LIN {X 0,Y 361.924,Z 605.401,A -85,B 0,C 180,E1 -12943.066,E2 -12943.066} C_VEL
LIN {X 0,Y 361.991,Z 605.395,A -85,B 0,C 180,E1 -12946.528,E2 -12946.528} C_VEL
LIN {X 0,Y 362.028,Z 605.391,A -85,B 0,C 180,E1 -12949.938,E2 -12949.938} C_VEL
LIN {X 0,Y 362.143,Z 605.376,A -85,B 0,C 180,E1 -12952.193,E2 -12952.193} C_VEL
LIN {X 0,Y 362.116,Z 605.378,A -85,B 0,C 180,E1 -12954.432,E2 -12954.432} C_VEL
LIN {X 0,Y 362.281,Z 605.357,A -85,B 0,C 180,E1 -12957.777,E2 -12957.777} C_VEL
LIN {X 0,Y 362.421,Z 605.339,A -85,B 0,C 180,E1 -12960.001,E2 -12960.001} C_VEL
LIN {X 0,Y 362.275,Z 605.357,A -85,B 0,C 180,E1 -12962.224,E2 -12962.224} C_VEL
LIN {X 0,Y 362.169,Z 605.369,A -85,B 0,C 180,E1 -12966.687,E2 -12966.687} C_VEL
LIN {X 0,Y 362.068,Z 605.384,A -85,B 0,C 180,E1 -12968.934,E2 -12968.934} C_VEL
LIN {X 0,Y 361.959,Z 605.395,A -85,B 0,C 180,E1 -12972.333,E2 -12972.333} C_VEL
LIN {X 0,Y 361.955,Z 605.398,A -85,B 0,C 180,E1 -12974.621,E2 -12974.621} C_VEL
LIN {X 0,Y 361.949,Z 605.397,A -85,B 0,C 180,E1 -12978.1,E2 -12978.1} C_VEL
LIN {X 0,Y 361.885,Z 605.403,A -85,B 0,C 180,E1 -12981.654,E2 -12981.654} C_VEL
LIN {X 0,Y 361.922,Z 605.398,A -85,B 0,C 180,E1 -12985.291,E2 -12985.291} C_VEL
LIN {X 0,Y 361.917,Z 605.399,A -85,B 0,C 180,E1 -12987.779,E2 -12987.779} C_VEL
LIN {X 0,Y 361.855,Z 605.403,A -85,B 0,C 180,E1 -12991.628,E2 -12991.628} C_VEL
LIN {X 0,Y 361.87,Z 605.404,A -85,B 0,C 180,E1 -12995.346,E2 -12995.346} C_VEL
LIN {X 0,Y 361.87,Z 605.406,A -85,B 0,C 180,E1 -12999.028,E2 -12999.028} C_VEL
LIN {X 0,Y 361.854,Z 605.41,A -85,B 0,C 180,E1 -13002.437,E2 -13002.437} C_VEL
LIN {X 0,Y 361.855,Z 605.41,A -85,B 0,C 180,E1 -13005.941,E2 -13005.941} C_VEL
LIN {X 0,Y 361.872,Z 605.412,A -85,B 0,C 180,E1 -13009.239,E2 -13009.239} C_VEL
LIN {X 0,Y 361.869,Z 605.41,A -85,B 0,C 180,E1 -13012.983,E2 -13012.983} C_VEL
LIN {X 0,Y 361.859,Z 605.415,A -85,B 0,C 180,E1 -13016.632,E2 -13016.632} C_VEL
LIN {X 0,Y 361.9,Z 605.535,A -85,B 0,C 180,E1 -13018.173,E2 -13018.173} C_VEL
LIN {X 0,Y 364.745,Z 617.624,A -85,B 0,C 180,E1 -13021.504,E2 -13021.504} C_VEL
LIN {X 0,Y 366.436,Z 626.629,A -85,B 0,C 180,E1 -13023.825,E2 -13023.825} C_VEL
LIN {X 0,Y 366.356,Z 630.226,A -85,B 0,C 180,E1 -13024.675,E2 -13024.675} C_VEL
LIN {X 0,Y 365,Z 642.315,A -85,B 0,C 180,E1 -13027.4,E2 -13027.4} C_VEL
LIN {X 0,Y 368.728,Z 663.081,A -85,B 0,C 180,E1 -13028.168,E2 -13028.168} C_VEL
LIN {X 0,Y 370.835,Z 679.65,A -85,B 0,C 180,E1 -13028.7,E2 -13028.7} C_VEL
LIN {X 0,Y 369.25,Z 751.918,A -85,B 0,C 180,E1 -13030.255,E2 -13030.255} C_VEL
LIN {X 0,Y 368.491,Z 765.438,A -85,B 0,C 180,E1 -13030.756,E2 -13030.756} C_VEL
LIN {X 0,Y 367.488,Z 778.333,A -85,B 0,C 180,E1 -13031.462,E2 -13031.462} C_VEL
LIN {X 0,Y 366.395,Z 790.927,A -85,B 0,C 180,E1 -13032.416,E2 -13032.416} C_VEL
LIN {X 0,Y 365.176,Z 802.216,A -85,B 0,C 180,E1 -13033.509,E2 -13033.509} C_VEL
LIN {X 0,Y 364.22,Z 811.35,A -85,B 0,C 180,E1 -13034.609,E2 -13034.609} C_VEL
LIN {X 0,Y 363.178,Z 820.833,A -85,B 0,C 180,E1 -13036.002,E2 -13036.002} C_VEL
LIN {X 0,Y 362.185,Z 830.004,A -85,B 0,C 180,E1 -13037.676,E2 -13037.676} C_VEL
LIN {X 0,Y 361.378,Z 837.416,A -85,B 0,C 180,E1 -13039.353,E2 -13039.353} C_VEL
LIN {X 0,Y 360.884,Z 843.38,A -85,B 0,C 180,E1 -13041.037,E2 -13041.037} C_VEL
LIN {X 0,Y 360.589,Z 848.087,A -85,B 0,C 180,E1 -13042.722,E2 -13042.722} C_VEL
LIN {X 0,Y 360.406,Z 851.68,A -85,B 0,C 180,E1 -13044.405,E2 -13044.405} C_VEL
LIN {X 0,Y 360.389,Z 853.485,A -85,B 0,C 180,E1 -13045.526,E2 -13045.526} C_VEL
LIN {X 0,Y 360.376,Z 855.852,A -85,B 0,C 180,E1 -13047.765,E2 -13047.765} C_VEL
LIN {X 0,Y 360.457,Z 856.421,A -85,B 0,C 180,E1 -13048.883,E2 -13048.883} C_VEL
LIN {X 0,Y 360.477,Z 856.542,A -85,B 0,C 180,E1 -13050,E2 -13050} C_VEL
LIN {X 0,Y 360.475,Z 856.264,A -85,B 0,C 180,E1 -13051.117,E2 -13051.117} C_VEL
LIN {X 0,Y 360.391,Z 855.583,A -85,B 0,C 180,E1 -13052.235,E2 -13052.235} C_VEL
LIN {X 0,Y 360.343,Z 854.477,A -85,B 0,C 180,E1 -13053.354,E2 -13053.354} C_VEL
LIN {X 0,Y 360.405,Z 852.916,A -85,B 0,C 180,E1 -13054.474,E2 -13054.474} C_VEL
LIN {X 0,Y 360.398,Z 850.122,A -85,B 0,C 180,E1 -13055.99,E2 -13055.99} C_VEL
LIN {X 0,Y 360.652,Z 845.489,A -85,B 0,C 180,E1 -13057.84,E2 -13057.84} C_VEL
LIN {X 0,Y 361.084,Z 838.99,A -85,B 0,C 180,E1 -13059.805,E2 -13059.805} C_VEL
LIN {X 0,Y 361.666,Z 831.869,A -85,B 0,C 180,E1 -13061.489,E2 -13061.489} C_VEL
LIN {X 0,Y 362.532,Z 822.949,A -85,B 0,C 180,E1 -13063.166,E2 -13063.166} C_VEL
LIN {X 0,Y 363.38,Z 813.8,A -85,B 0,C 180,E1 -13064.562,E2 -13064.562} C_VEL
LIN {X 0,Y 364.28,Z 803.709,A -85,B 0,C 180,E1 -13065.813,E2 -13065.813} C_VEL
LIN {X 0,Y 365.348,Z 792.51,A -85,B 0,C 180,E1 -13066.914,E2 -13066.914} C_VEL
LIN {X 0,Y 366.353,Z 779.984,A -85,B 0,C 180,E1 -13067.874,E2 -13067.874} C_VEL
LIN {X 0,Y 367.228,Z 767.268,A -85,B 0,C 180,E1 -13068.588,E2 -13068.588} C_VEL
LIN {X 0,Y 367.908,Z 753.937,A -85,B 0,C 180,E1 -13069.094,E2 -13069.094} C_VEL
LIN {X 0,Y 368.878,Z 705.145,A -85,B 0,C 180,E1 -13070.137,E2 -13070.137} C_VEL
LIN {X 0,Y 369.232,Z 677.948,A -85,B 0,C 180,E1 -13070.712,E2 -13070.712} C_VEL
LIN {X 0,Y 364.358,Z 643.946,A -85,B 0,C 180,E1 -13071.759,E2 -13071.759} C_VEL
LIN {X 0,Y 366.056,Z 626.823,A -85,B 0,C 180,E1 -13075.528,E2 -13075.528} C_VEL
LIN {X 0,Y 364.723,Z 618.389,A -85,B 0,C 180,E1 -13077.546,E2 -13077.546} C_VEL
LIN {X 0,Y 361.886,Z 605.407,A -85,B 0,C 180,E1 -13080.822,E2 -13080.822} C_VEL
LIN {X 0,Y 361.854,Z 605.412,A -85,B 0,C 180,E1 -13084.279,E2 -13084.279} C_VEL
LIN {X 0,Y 361.865,Z 605.406,A -85,B 0,C 180,E1 -13087.222,E2 -13087.222} C_VEL
LIN {X 0,Y 361.871,Z 605.409,A -85,B 0,C 180,E1 -13090.761,E2 -13090.761} C_VEL
LIN {X 0,Y 361.863,Z 605.41,A -85,B 0,C 180,E1 -13094.36,E2 -13094.36} C_VEL
LIN {X 0,Y 361.854,Z 605.407,A -85,B 0,C 180,E1 -13097.563,E2 -13097.563} C_VEL
LIN {X 0,Y 361.872,Z 605.409,A -85,B 0,C 180,E1 -13100.971,E2 -13100.971} C_VEL
LIN {X 0,Y 361.871,Z 605.41,A -85,B 0,C 180,E1 -13104.654,E2 -13104.654} C_VEL
LIN {X 0,Y 361.855,Z 605.408,A -85,B 0,C 180,E1 -13108.372,E2 -13108.372} C_VEL
LIN {X 0,Y 361.917,Z 605.399,A -85,B 0,C 180,E1 -13112.221,E2 -13112.221} C_VEL
LIN {X 0,Y 361.921,Z 605.402,A -85,B 0,C 180,E1 -13114.709,E2 -13114.709} C_VEL
LIN {X 0,Y 361.855,Z 605.407,A -85,B 0,C 180,E1 -13118.344,E2 -13118.344} C_VEL
LIN {X 0,Y 361.961,Z 605.394,A -85,B 0,C 180,E1 -13122.061,E2 -13122.061} C_VEL
LIN {X 0,Y 361.99,Z 605.39,A -85,B 0,C 180,E1 -13126.101,E2 -13126.101} C_VEL
LIN {X 0,Y 362.024,Z 605.387,A -85,B 0,C 180,E1 -13129.937,E2 -13129.937} C_VEL
LIN {X 0,Y 362.155,Z 605.376,A -85,B 0,C 180,E1 -13133.313,E2 -13133.313} C_VEL
LIN {X 0,Y 362.275,Z 605.357,A -85,B 0,C 180,E1 -13137.776,E2 -13137.776} C_VEL
LIN {X 0,Y 362.421,Z 605.338,A -85,B 0,C 180,E1 -13139.999,E2 -13139.999} C_VEL
LIN {X 0,Y 362.275,Z 605.355,A -85,B 0,C 180,E1 -13142.223,E2 -13142.223} C_VEL
LIN {X 0,Y 362.159,Z 605.369,A -85,B 0,C 180,E1 -13146.686,E2 -13146.686} C_VEL
LIN {X 0,Y 362.024,Z 605.388,A -85,B 0,C 180,E1 -13150.062,E2 -13150.062} C_VEL
LIN {X 0,Y 361.989,Z 605.395,A -85,B 0,C 180,E1 -13153.898,E2 -13153.898} C_VEL
LIN {X 0,Y 361.958,Z 605.399,A -85,B 0,C 180,E1 -13157.938,E2 -13157.938} C_VEL
LIN {X 0,Y 361.883,Z 605.408,A -85,B 0,C 180,E1 -13161.653,E2 -13161.653} C_VEL
LIN {X 0,Y 361.919,Z 605.4,A -85,B 0,C 180,E1 -13165.29,E2 -13165.29} C_VEL
LIN {X 0,Y 361.914,Z 605.404,A -85,B 0,C 180,E1 -13167.778,E2 -13167.778} C_VEL
LIN {X 0,Y 361.851,Z 605.41,A -85,B 0,C 180,E1 -13171.627,E2 -13171.627} C_VEL
LIN {X 0,Y 361.866,Z 605.406,A -85,B 0,C 180,E1 -13175.345,E2 -13175.345} C_VEL
LIN {X 0,Y 361.867,Z 605.405,A -85,B 0,C 180,E1 -13179.028,E2 -13179.028} C_VEL
LIN {X 0,Y 361.882,Z 605.408,A -85,B 0,C 180,E1 -13182.441,E2 -13182.441} C_VEL
LIN {X 0,Y 361.859,Z 605.407,A -85,B 0,C 180,E1 -13185.639,E2 -13185.639} C_VEL
LIN {X 0,Y 361.865,Z 605.406,A -85,B 0,C 180,E1 -13189.238,E2 -13189.238} C_VEL
LIN {X 0,Y 361.866,Z 605.407,A -85,B 0,C 180,E1 -13192.983,E2 -13192.983} C_VEL
LIN {X 0,Y 361.853,Z 605.412,A -85,B 0,C 180,E1 -13196.631,E2 -13196.631} C_VEL
LIN {X 0,Y 361.867,Z 605.405,A -85,B 0,C 180,E1 -13199.672,E2 -13199.672} C_VEL
LIN {X 0,Y 361.949,Z 605.395,A -85,B 0,C 180,E1 -13203.475,E2 -13203.475} C_VEL
LIN {X 0,Y 361.887,Z 605.405,A -85,B 0,C 180,E1 -13207.145,E2 -13207.145} C_VEL
LIN {X 0,Y 361.902,Z 605.408,A -85,B 0,C 180,E1 -13210.724,E2 -13210.724} C_VEL
LIN {X 0,Y 361.929,Z 605.401,A -85,B 0,C 180,E1 -13213.066,E2 -13213.066} C_VEL
LIN {X 0,Y 361.995,Z 605.393,A -85,B 0,C 180,E1 -13216.528,E2 -13216.528} C_VEL
LIN {X 0,Y 362.028,Z 605.385,A -85,B 0,C 180,E1 -13219.938,E2 -13219.938} C_VEL
LIN {X 0,Y 362.157,Z 605.372,A -85,B 0,C 180,E1 -13223.314,E2 -13223.314} C_VEL
LIN {X 0,Y 362.28,Z 605.354,A -85,B 0,C 180,E1 -13227.776,E2 -13227.776} C_VEL
LIN {X 0,Y 362.425,Z 605.336,A -85,B 0,C 180,E1 -13230,E2 -13230} C_VEL
LIN {X 0,Y 362.28,Z 605.354,A -85,B 0,C 180,E1 -13232.224,E2 -13232.224} C_VEL
LIN {X 0,Y 362.158,Z 605.371,A -85,B 0,C 180,E1 -13236.686,E2 -13236.686} C_VEL
LIN {X 0,Y 362.028,Z 605.385,A -85,B 0,C 180,E1 -13240.062,E2 -13240.062} C_VEL
LIN {X 0,Y 361.994,Z 605.391,A -85,B 0,C 180,E1 -13243.899,E2 -13243.899} C_VEL
LIN {X 0,Y 361.963,Z 605.399,A -85,B 0,C 180,E1 -13247.938,E2 -13247.938} C_VEL
LIN {X 0,Y 361.907,Z 605.413,A -85,B 0,C 180,E1 -13251.574,E2 -13251.574} C_VEL
LIN {X 0,Y 363.096,Z 611.348,A -85,B 0,C 180,E1 -13253.302,E2 -13253.302} C_VEL
LIN {X 0,Y 367.795,Z 625.296,A -85,B 0,C 180,E1 -13253.875,E2 -13253.875} C_VEL
LIN {X 0,Y 369.865,Z 635.286,A -85,B 0,C 180,E1 -13254.208,E2 -13254.208} C_VEL
LIN {X 0,Y 368.159,Z 718.4,A -85,B 0,C 180,E1 -13255.954,E2 -13255.954} C_VEL
LIN {X 0,Y 367.654,Z 732.266,A -85,B 0,C 180,E1 -13256.482,E2 -13256.482} C_VEL
LIN {X 0,Y 366.978,Z 745.105,A -85,B 0,C 180,E1 -13257.208,E2 -13257.208} C_VEL
LIN {X 0,Y 366.657,Z 749.389,A -85,B 0,C 180,E1 -13257.503,E2 -13257.503} C_VEL
LIN {X 0,Y 365.652,Z 754.736,A -85,B 0,C 180,E1 -13257.89,E2 -13257.89} C_VEL
LIN {X 0,Y 362.237,Z 763.117,A -85,B 0,C 180,E1 -13258.53,E2 -13258.53} C_VEL
LIN {X 0,Y 358.758,Z 771.115,A -85,B 0,C 180,E1 -13259.271,E2 -13259.271} C_VEL
LIN {X 0,Y 357.633,Z 775.748,A -85,B 0,C 180,E1 -13259.82,E2 -13259.82} C_VEL
LIN {X 0,Y 356.659,Z 786.017,A -85,B 0,C 180,E1 -13261.313,E2 -13261.313} C_VEL
LIN {X 0,Y 355.739,Z 794.802,A -85,B 0,C 180,E1 -13262.907,E2 -13262.907} C_VEL
LIN {X 0,Y 354.896,Z 802.812,A -85,B 0,C 180,E1 -13264.727,E2 -13264.727} C_VEL
LIN {X 0,Y 354.312,Z 809.044,A -85,B 0,C 180,E1 -13266.516,E2 -13266.516} C_VEL
LIN {X 0,Y 353.912,Z 813.113,A -85,B 0,C 180,E1 -13267.994,E2 -13267.994} C_VEL
LIN {X 0,Y 353.615,Z 816.393,A -85,B 0,C 180,E1 -13269.492,E2 -13269.492} C_VEL
LIN {X 0,Y 353.393,Z 818.933,A -85,B 0,C 180,E1 -13271.015,E2 -13271.015} C_VEL
LIN {X 0,Y 353.232,Z 820.757,A -85,B 0,C 180,E1 -13272.596,E2 -13272.596} C_VEL
LIN {X 0,Y 353.126,Z 821.787,A -85,B 0,C 180,E1 -13274.236,E2 -13274.236} C_VEL
LIN {X 0,Y 353.144,Z 821.99,A -85,B 0,C 180,E1 -13275.851,E2 -13275.851} C_VEL
LIN {X 0,Y 353.24,Z 821.42,A -85,B 0,C 180,E1 -13277.433,E2 -13277.433} C_VEL
LIN {X 0,Y 353.439,Z 820.008,A -85,B 0,C 180,E1 -13279.078,E2 -13279.078} C_VEL
LIN {X 0,Y 353.768,Z 817.614,A -85,B 0,C 180,E1 -13280.783,E2 -13280.783} C_VEL
LIN {X 0,Y 354.179,Z 814.121,A -85,B 0,C 180,E1 -13282.533,E2 -13282.533} C_VEL
LIN {X 0,Y 354.739,Z 809.363,A -85,B 0,C 180,E1 -13284.317,E2 -13284.317} C_VEL
LIN {X 0,Y 355.514,Z 803.146,A -85,B 0,C 180,E1 -13286.125,E2 -13286.125} C_VEL
LIN {X 0,Y 356.506,Z 795.17,A -85,B 0,C 180,E1 -13287.958,E2 -13287.958} C_VEL
LIN {X 0,Y 357.704,Z 786.246,A -85,B 0,C 180,E1 -13289.573,E2 -13289.573} C_VEL
LIN {X 0,Y 358.859,Z 775.956,A -85,B 0,C 180,E1 -13291.071,E2 -13291.071} C_VEL
LIN {X 0,Y 359.92,Z 766.222,A -85,B 0,C 180,E1 -13292.213,E2 -13292.213} C_VEL
LIN {X 0,Y 361.008,Z 755.205,A -85,B 0,C 180,E1 -13293.245,E2 -13293.245} C_VEL
LIN {X 0,Y 362.006,Z 742.249,A -85,B 0,C 180,E1 -13294.177,E2 -13294.177} C_VEL
LIN {X 0,Y 362.656,Z 729.115,A -85,B 0,C 180,E1 -13294.863,E2 -13294.863} C_VEL
LIN {X 0,Y 363.21,Z 715.436,A -85,B 0,C 180,E1 -13295.309,E2 -13295.309} C_VEL
LIN {X 0,Y 365.063,Z 636.901,A -85,B 0,C 180,E1 -13297.028,E2 -13297.028} C_VEL
LIN {X 0,Y 363.354,Z 630.119,A -85,B 0,C 180,E1 -13297.318,E2 -13297.318} C_VEL
LIN {X 0,Y 356.414,Z 613.512,A -85,B 0,C 180,E1 -13298.298,E2 -13298.298} C_VEL
LIN {X 0,Y 354.882,Z 606.281,A -85,B 0,C 180,E1 -13300.778,E2 -13300.778} C_VEL
LIN {X 0,Y 354.881,Z 606.28,A -85,B 0,C 180,E1 -13303.904,E2 -13303.904} C_VEL
LIN {X 0,Y 354.918,Z 606.275,A -85,B 0,C 180,E1 -13307.42,E2 -13307.42} C_VEL
LIN {X 0,Y 355.12,Z 606.251,A -85,B 0,C 180,E1 -13311.69,E2 -13311.69} C_VEL
LIN {X 0,Y 355.09,Z 606.253,A -85,B 0,C 180,E1 -13314.321,E2 -13314.321} C_VEL
LIN {X 0,Y 355.245,Z 606.233,A -85,B 0,C 180,E1 -13317.733,E2 -13317.733} C_VEL
LIN {X 0,Y 355.39,Z 606.215,A -85,B 0,C 180,E1 -13320.001,E2 -13320.001} C_VEL
LIN {X 0,Y 355.238,Z 606.234,A -85,B 0,C 180,E1 -13322.268,E2 -13322.268} C_VEL
LIN {X 0,Y 355.135,Z 606.245,A -85,B 0,C 180,E1 -13326.82,E2 -13326.82} C_VEL
LIN {X 0,Y 355.009,Z 606.261,A -85,B 0,C 180,E1 -13329.113,E2 -13329.113} C_VEL
LIN {X 0,Y 354.919,Z 606.272,A -85,B 0,C 180,E1 -13332.582,E2 -13332.582} C_VEL
LIN {X 0,Y 354.883,Z 606.272,A -85,B 0,C 180,E1 -13336.097,E2 -13336.097} C_VEL
LIN {X 0,Y 354.895,Z 606.277,A -85,B 0,C 180,E1 -13338.473,E2 -13338.473} C_VEL
LIN {X 0,Y 354.828,Z 606.281,A -85,B 0,C 180,E1 -13342.107,E2 -13342.107} C_VEL
LIN {X 0,Y 354.894,Z 606.271,A -85,B 0,C 180,E1 -13345.828,E2 -13345.828} C_VEL
LIN {X 0,Y 354.85,Z 606.28,A -85,B 0,C 180,E1 -13349.68,E2 -13349.68} C_VEL
LIN {X 0,Y 354.827,Z 606.284,A -85,B 0,C 180,E1 -13353.683,E2 -13353.683} C_VEL
LIN {X 0,Y 354.795,Z 606.287,A -85,B 0,C 180,E1 -13356.46,E2 -13356.46} C_VEL
LIN {X 0,Y 354.821,Z 606.289,A -85,B 0,C 180,E1 -13359.425,E2 -13359.425} C_VEL
LIN {X 0,Y 354.802,Z 606.29,A -85,B 0,C 180,E1 -13362.871,E2 -13362.871} C_VEL
LIN {X 0,Y 354.8,Z 606.289,A -85,B 0,C 180,E1 -13366.11,E2 -13366.11} C_VEL
LIN {X 0,Y 354.823,Z 606.289,A -85,B 0,C 180,E1 -13369.185,E2 -13369.185} C_VEL
LIN {X 0,Y 354.809,Z 606.289,A -85,B 0,C 180,E1 -13372.403,E2 -13372.403} C_VEL
LIN {X 0,Y 354.812,Z 606.289,A -85,B 0,C 180,E1 -13374.942,E2 -13374.942} C_VEL
LIN {X 0,Y 354.841,Z 606.45,A -85,B 0,C 180,E1 -13377.673,E2 -13377.673} C_VEL
LIN {X 0,Y 357.556,Z 617.727,A -85,B 0,C 180,E1 -13380.892,E2 -13380.892} C_VEL
LIN {X 0,Y 359.341,Z 626.618,A -85,B 0,C 180,E1 -13383.268,E2 -13383.268} C_VEL
LIN {X 0,Y 359.643,Z 630.28,A -85,B 0,C 180,E1 -13384.184,E2 -13384.184} C_VEL
LIN {X 0,Y 358.239,Z 641.954,A -85,B 0,C 180,E1 -13386.88,E2 -13386.88} C_VEL
LIN {X 0,Y 362.078,Z 662.796,A -85,B 0,C 180,E1 -13387.683,E2 -13387.683} C_VEL
LIN {X 0,Y 364.348,Z 680.292,A -85,B 0,C 180,E1 -13388.262,E2 -13388.262} C_VEL
LIN {X 0,Y 362.68,Z 751.869,A -85,B 0,C 180,E1 -13389.845,E2 -13389.845} C_VEL
LIN {X 0,Y 361.821,Z 765.979,A -85,B 0,C 180,E1 -13390.387,E2 -13390.387} C_VEL
LIN {X 0,Y 360.792,Z 778.534,A -85,B 0,C 180,E1 -13391.105,E2 -13391.105} C_VEL
LIN {X 0,Y 359.64,Z 791.01,A -85,B 0,C 180,E1 -13392.075,E2 -13392.075} C_VEL
LIN {X 0,Y 358.369,Z 802.22,A -85,B 0,C 180,E1 -13393.187,E2 -13393.187} C_VEL
LIN {X 0,Y 357.204,Z 812.652,A -85,B 0,C 180,E1 -13394.497,E2 -13394.497} C_VEL
LIN {X 0,Y 356.123,Z 822.366,A -85,B 0,C 180,E1 -13396.01,E2 -13396.01} C_VEL
LIN {X 0,Y 355.059,Z 831.213,A -85,B 0,C 180,E1 -13397.715,E2 -13397.715} C_VEL
LIN {X 0,Y 354.281,Z 838.29,A -85,B 0,C 180,E1 -13399.427,E2 -13399.427} C_VEL
LIN {X 0,Y 353.698,Z 844.814,A -85,B 0,C 180,E1 -13401.43,E2 -13401.43} C_VEL
LIN {X 0,Y 353.424,Z 849.109,A -85,B 0,C 180,E1 -13403.148,E2 -13403.148} C_VEL
LIN {X 0,Y 353.332,Z 851.39,A -85,B 0,C 180,E1 -13404.292,E2 -13404.292} C_VEL
LIN {X 0,Y 353.301,Z 853.18,A -85,B 0,C 180,E1 -13405.436,E2 -13405.436} C_VEL
LIN {X 0,Y 353.265,Z 854.556,A -85,B 0,C 180,E1 -13406.578,E2 -13406.578} C_VEL
LIN {X 0,Y 353.277,Z 855.53,A -85,B 0,C 180,E1 -13407.72,E2 -13407.72} C_VEL
LIN {X 0,Y 353.36,Z 856.079,A -85,B 0,C 180,E1 -13408.86,E2 -13408.86} C_VEL
LIN {X 0,Y 353.414,Z 856.191,A -85,B 0,C 180,E1 -13410,E2 -13410} C_VEL
LIN {X 0,Y 353.393,Z 855.901,A -85,B 0,C 180,E1 -13411.139,E2 -13411.139} C_VEL
LIN {X 0,Y 353.293,Z 855.208,A -85,B 0,C 180,E1 -13412.28,E2 -13412.28} C_VEL
LIN {X 0,Y 353.263,Z 854.078,A -85,B 0,C 180,E1 -13413.422,E2 -13413.422} C_VEL
LIN {X 0,Y 353.292,Z 851.575,A -85,B 0,C 180,E1 -13415.136,E2 -13415.136} C_VEL
LIN {X 0,Y 353.418,Z 848.027,A -85,B 0,C 180,E1 -13416.852,E2 -13416.852} C_VEL
LIN {X 0,Y 353.693,Z 843.343,A -85,B 0,C 180,E1 -13418.57,E2 -13418.57} C_VEL
LIN {X 0,Y 354.21,Z 836.241,A -85,B 0,C 180,E1 -13420.575,E2 -13420.575} C_VEL
LIN {X 0,Y 354.963,Z 828.548,A -85,B 0,C 180,E1 -13422.289,E2 -13422.289} C_VEL
LIN {X 0,Y 355.741,Z 820.66,A -85,B 0,C 180,E1 -13423.713,E2 -13423.713} C_VEL
LIN {X 0,Y 356.612,Z 811.228,A -85,B 0,C 180,E1 -13425.107,E2 -13425.107} C_VEL
LIN {X 0,Y 357.702,Z 800.324,A -85,B 0,C 180,E1 -13426.405,E2 -13426.405} C_VEL
LIN {X 0,Y 358.707,Z 790.038,A -85,B 0,C 180,E1 -13427.384,E2 -13427.384} C_VEL
LIN {X 0,Y 359.635,Z 777.841,A -85,B 0,C 180,E1 -13428.294,E2 -13428.294} C_VEL
LIN {X 0,Y 360.573,Z 764.394,A -85,B 0,C 180,E1 -13429.018,E2 -13429.018} C_VEL
LIN {X 0,Y 361.162,Z 752.079,A -85,B 0,C 180,E1 -13429.465,E2 -13429.465} C_VEL
LIN {X 0,Y 362.52,Z 678.883,A -85,B 0,C 180,E1 -13431.041,E2 -13431.041} C_VEL
LIN {X 0,Y 357.497,Z 643.703,A -85,B 0,C 180,E1 -13432.135,E2 -13432.135} C_VEL
LIN {X 0,Y 359.102,Z 627.366,A -85,B 0,C 180,E1 -13435.806,E2 -13435.806} C_VEL
LIN {X 0,Y 357.334,Z 617.793,A -85,B 0,C 180,E1 -13438.165,E2 -13438.165} C_VEL
LIN {X 0,Y 354.827,Z 606.287,A -85,B 0,C 180,E1 -13441.159,E2 -13441.159} C_VEL
LIN {X 0,Y 354.812,Z 606.285,A -85,B 0,C 180,E1 -13445.058,E2 -13445.058} C_VEL
LIN {X 0,Y 354.807,Z 606.286,A -85,B 0,C 180,E1 -13447.881,E2 -13447.881} C_VEL
LIN {X 0,Y 354.815,Z 606.285,A -85,B 0,C 180,E1 -13451.176,E2 -13451.176} C_VEL
LIN {X 0,Y 354.821,Z 606.288,A -85,B 0,C 180,E1 -13454.515,E2 -13454.515} C_VEL
LIN {X 0,Y 354.81,Z 606.284,A -85,B 0,C 180,E1 -13457.664,E2 -13457.664} C_VEL
LIN {X 0,Y 354.834,Z 606.287,A -85,B 0,C 180,E1 -13460.668,E2 -13460.668} C_VEL
LIN {X 0,Y 354.819,Z 606.285,A -85,B 0,C 180,E1 -13464.3,E2 -13464.3} C_VEL
LIN {X 0,Y 354.794,Z 606.287,A -85,B 0,C 180,E1 -13467.667,E2 -13467.667} C_VEL
LIN {X 0,Y 354.864,Z 606.281,A -85,B 0,C 180,E1 -13470.62,E2 -13470.62} C_VEL
LIN {X 0,Y 354.893,Z 606.274,A -85,B 0,C 180,E1 -13474.172,E2 -13474.172} C_VEL
LIN {X 0,Y 354.81,Z 606.284,A -85,B 0,C 180,E1 -13477.892,E2 -13477.892} C_VEL
LIN {X 0,Y 354.916,Z 606.272,A -85,B 0,C 180,E1 -13481.891,E2 -13481.891} C_VEL
LIN {X 0,Y 354.935,Z 606.269,A -85,B 0,C 180,E1 -13485.981,E2 -13485.981} C_VEL
LIN {X 0,Y 354.97,Z 606.266,A -85,B 0,C 180,E1 -13489.735,E2 -13489.735} C_VEL
LIN {X 0,Y 355.119,Z 606.251,A -85,B 0,C 180,E1 -13493.18,E2 -13493.18} C_VEL
LIN {X 0,Y 355.238,Z 606.234,A -85,B 0,C 180,E1 -13497.732,E2 -13497.732} C_VEL
LIN {X 0,Y 355.39,Z 606.214,A -85,B 0,C 180,E1 -13499.999,E2 -13499.999} C_VEL
LIN {X 0,Y 355.238,Z 606.231,A -85,B 0,C 180,E1 -13502.267,E2 -13502.267} C_VEL
LIN {X 0,Y 355.122,Z 606.246,A -85,B 0,C 180,E1 -13506.819,E2 -13506.819} C_VEL
LIN {X 0,Y 354.971,Z 606.265,A -85,B 0,C 180,E1 -13510.264,E2 -13510.264} C_VEL
LIN {X 0,Y 354.934,Z 606.272,A -85,B 0,C 180,E1 -13514.018,E2 -13514.018} C_VEL
LIN {X 0,Y 354.914,Z 606.275,A -85,B 0,C 180,E1 -13518.108,E2 -13518.108} C_VEL
LIN {X 0,Y 354.826,Z 606.286,A -85,B 0,C 180,E1 -13522.106,E2 -13522.106} C_VEL
LIN {X 0,Y 354.891,Z 606.28,A -85,B 0,C 180,E1 -13525.827,E2 -13525.827} C_VEL
LIN {X 0,Y 354.846,Z 606.283,A -85,B 0,C 180,E1 -13529.679,E2 -13529.679} C_VEL
LIN {X 0,Y 354.823,Z 606.285,A -85,B 0,C 180,E1 -13533.682,E2 -13533.682} C_VEL
LIN {X 0,Y 354.792,Z 606.29,A -85,B 0,C 180,E1 -13536.459,E2 -13536.459} C_VEL
LIN {X 0,Y 354.816,Z 606.284,A -85,B 0,C 180,E1 -13539.424,E2 -13539.424} C_VEL
LIN {X 0,Y 354.83,Z 606.283,A -85,B 0,C 180,E1 -13542.876,E2 -13542.876} C_VEL
LIN {X 0,Y 354.799,Z 606.291,A -85,B 0,C 180,E1 -13546.11,E2 -13546.11} C_VEL
LIN {X 0,Y 354.817,Z 606.284,A -85,B 0,C 180,E1 -13549.184,E2 -13549.184} C_VEL
LIN {X 0,Y 354.806,Z 606.292,A -85,B 0,C 180,E1 -13552.402,E2 -13552.402} C_VEL
LIN {X 0,Y 354.806,Z 606.287,A -85,B 0,C 180,E1 -13554.941,E2 -13554.941} C_VEL
LIN {X 0,Y 354.788,Z 606.293,A -85,B 0,C 180,E1 -13558.405,E2 -13558.405} C_VEL
LIN {X 0,Y 354.841,Z 606.281,A -85,B 0,C 180,E1 -13561.619,E2 -13561.619} C_VEL
LIN {X 0,Y 354.894,Z 606.276,A -85,B 0,C 180,E1 -13564.173,E2 -13564.173} C_VEL
LIN {X 0,Y 354.831,Z 606.282,A -85,B 0,C 180,E1 -13567.894,E2 -13567.894} C_VEL
LIN {X 0,Y 354.918,Z 606.271,A -85,B 0,C 180,E1 -13571.892,E2 -13571.892} C_VEL
LIN {X 0,Y 354.939,Z 606.268,A -85,B 0,C 180,E1 -13575.981,E2 -13575.981} C_VEL
LIN {X 0,Y 354.975,Z 606.264,A -85,B 0,C 180,E1 -13579.736,E2 -13579.736} C_VEL
LIN {X 0,Y 355.122,Z 606.25,A -85,B 0,C 180,E1 -13583.181,E2 -13583.181} C_VEL
LIN {X 0,Y 355.243,Z 606.231,A -85,B 0,C 180,E1 -13587.732,E2 -13587.732} C_VEL
LIN {X 0,Y 355.395,Z 606.212,A -85,B 0,C 180,E1 -13590,E2 -13590} C_VEL
LIN {X 0,Y 355.243,Z 606.231,A -85,B 0,C 180,E1 -13592.268,E2 -13592.268} C_VEL
LIN {X 0,Y 355.121,Z 606.248,A -85,B 0,C 180,E1 -13596.819,E2 -13596.819} C_VEL
LIN {X 0,Y 354.975,Z 606.264,A -85,B 0,C 180,E1 -13600.264,E2 -13600.264} C_VEL
LIN {X 0,Y 354.939,Z 606.269,A -85,B 0,C 180,E1 -13604.019,E2 -13604.019} C_VEL
LIN {X 0,Y 354.918,Z 606.276,A -85,B 0,C 180,E1 -13608.108,E2 -13608.108} C_VEL
LIN {X 0,Y 354.86,Z 606.284,A -85,B 0,C 180,E1 -13611.304,E2 -13611.304} C_VEL
LIN {X 0,Y 355.901,Z 611.442,A -85,B 0,C 180,E1 -13612.877,E2 -13612.877} C_VEL
LIN {X 0,Y 361.408,Z 627.849,A -85,B 0,C 180,E1 -13613.578,E2 -13613.578} C_VEL
LIN {X 0,Y 363.157,Z 636.67,A -85,B 0,C 180,E1 -13613.874,E2 -13613.874} C_VEL
LIN {X 0,Y 361.371,Z 718.839,A -85,B 0,C 180,E1 -13615.637,E2 -13615.637} C_VEL
LIN {X 0,Y 360.838,Z 732.774,A -85,B 0,C 180,E1 -13616.18,E2 -13616.18} C_VEL
LIN {X 0,Y 360.153,Z 745.32,A -85,B 0,C 180,E1 -13616.902,E2 -13616.902} C_VEL
LIN {X 0,Y 359.286,Z 757.382,A -85,B 0,C 180,E1 -13617.84,E2 -13617.84} C_VEL
LIN {X 0,Y 358.347,Z 768.268,A -85,B 0,C 180,E1 -13618.919,E2 -13618.919} C_VEL
LIN {X 0,Y 357.633,Z 775.748,A -85,B 0,C 180,E1 -13619.82,E2 -13619.82} C_VEL
LIN {X 0,Y 356.519,Z 780.296,A -85,B 0,C 180,E1 -13620.411,E2 -13620.411} C_VEL
LIN {X 0,Y 353.026,Z 787.328,A -85,B 0,C 180,E1 -13621.396,E2 -13621.396} C_VEL
LIN {X 0,Y 349.544,Z 793.824,A -85,B 0,C 180,E1 -13622.477,E2 -13622.477} C_VEL
LIN {X 0,Y 348.454,Z 797.459,A -85,B 0,C 180,E1 -13623.21,E2 -13623.21} C_VEL
LIN {X 0,Y 347.766,Z 804.068,A -85,B 0,C 180,E1 -13624.812,E2 -13624.812} C_VEL
LIN {X 0,Y 347.194,Z 810.145,A -85,B 0,C 180,E1 -13626.664,E2 -13626.664} C_VEL
LIN {X 0,Y 346.771,Z 814.439,A -85,B 0,C 180,E1 -13628.324,E2 -13628.324} C_VEL
LIN {X 0,Y 346.37,Z 818.538,A -85,B 0,C 180,E1 -13630.487,E2 -13630.487} C_VEL
LIN {X 0,Y 346.174,Z 820.567,A -85,B 0,C 180,E1 -13632.063,E2 -13632.063} C_VEL
LIN {X 0,Y 346.055,Z 821.864,A -85,B 0,C 180,E1 -13633.668,E2 -13633.668} C_VEL
LIN {X 0,Y 346.022,Z 822.376,A -85,B 0,C 180,E1 -13635.305,E2 -13635.305} C_VEL
LIN {X 0,Y 346.101,Z 822.059,A -85,B 0,C 180,E1 -13636.971,E2 -13636.971} C_VEL
LIN {X 0,Y 346.284,Z 820.895,A -85,B 0,C 180,E1 -13638.67,E2 -13638.67} C_VEL
LIN {X 0,Y 346.606,Z 818.807,A -85,B 0,C 180,E1 -13640.398,E2 -13640.398} C_VEL
LIN {X 0,Y 347.12,Z 814.772,A -85,B 0,C 180,E1 -13642.599,E2 -13642.599} C_VEL
LIN {X 0,Y 347.756,Z 809.944,A -85,B 0,C 180,E1 -13644.478,E2 -13644.478} C_VEL
LIN {X 0,Y 348.605,Z 803.344,A -85,B 0,C 180,E1 -13646.436,E2 -13646.436} C_VEL
LIN {X 0,Y 349.672,Z 795.361,A -85,B 0,C 180,E1 -13648.3,E2 -13648.3} C_VEL
LIN {X 0,Y 350.958,Z 786.31,A -85,B 0,C 180,E1 -13649.959,E2 -13649.959} C_VEL
LIN {X 0,Y 352.127,Z 776.456,A -85,B 0,C 180,E1 -13651.421,E2 -13651.421} C_VEL
LIN {X 0,Y 353.277,Z 766.498,A -85,B 0,C 180,E1 -13652.611,E2 -13652.611} C_VEL
LIN {X 0,Y 354.479,Z 754.537,A -85,B 0,C 180,E1 -13653.736,E2 -13653.736} C_VEL
LIN {X 0,Y 355.466,Z 742.161,A -85,B 0,C 180,E1 -13654.629,E2 -13654.629} C_VEL
LIN {X 0,Y 356.115,Z 729.259,A -85,B 0,C 180,E1 -13655.308,E2 -13655.308} C_VEL
LIN {X 0,Y 356.69,Z 716.293,A -85,B 0,C 180,E1 -13655.738,E2 -13655.738} C_VEL
LIN {X 0,Y 358.75,Z 638.622,A -85,B 0,C 180,E1 -13657.467,E2 -13657.467} C_VEL
LIN {X 0,Y 357.182,Z 632.506,A -85,B 0,C 180,E1 -13657.743,E2 -13657.743} C_VEL
LIN {X 0,Y 350.418,Z 616.665,A -85,B 0,C 180,E1 -13658.705,E2 -13658.705} C_VEL
LIN {X 0,Y 349.271,Z 613.867,A -85,B 0,C 180,E1 -13658.92,E2 -13658.92} C_VEL
LIN {X 0,Y 347.839,Z 607.157,A -85,B 0,C 180,E1 -13661.342,E2 -13661.342} C_VEL
LIN {X 0,Y 347.857,Z 607.156,A -85,B 0,C 180,E1 -13664.773,E2 -13664.773} C_VEL
LIN {X 0,Y 347.882,Z 607.154,A -85,B 0,C 180,E1 -13668.345,E2 -13668.345} C_VEL
LIN {X 0,Y 348.066,Z 607.13,A -85,B 0,C 180,E1 -13671.875,E2 -13671.875} C_VEL
LIN {X 0,Y 348.064,Z 607.129,A -85,B 0,C 180,E1 -13674.206,E2 -13674.206} C_VEL
LIN {X 0,Y 348.209,Z 607.11,A -85,B 0,C 180,E1 -13677.687,E2 -13677.687} C_VEL
LIN {X 0,Y 348.36,Z 607.091,A -85,B 0,C 180,E1 -13680.001,E2 -13680.001} C_VEL
LIN {X 0,Y 348.201,Z 607.11,A -85,B 0,C 180,E1 -13682.314,E2 -13682.314} C_VEL
LIN {X 0,Y 348.102,Z 607.121,A -85,B 0,C 180,E1 -13686.958,E2 -13686.958} C_VEL
LIN {X 0,Y 347.962,Z 607.137,A -85,B 0,C 180,E1 -13689.299,E2 -13689.299} C_VEL
LIN {X 0,Y 347.887,Z 607.147,A -85,B 0,C 180,E1 -13692.84,E2 -13692.84} C_VEL
LIN {X 0,Y 347.832,Z 607.151,A -85,B 0,C 180,E1 -13696.432,E2 -13696.432} C_VEL
LIN {X 0,Y 347.844,Z 607.153,A -85,B 0,C 180,E1 -13698.861,E2 -13698.861} C_VEL
LIN {X 0,Y 347.768,Z 607.16,A -85,B 0,C 180,E1 -13702.58,E2 -13702.58} C_VEL
LIN {X 0,Y 347.807,Z 607.157,A -85,B 0,C 180,E1 -13705.109,E2 -13705.109} C_VEL
LIN {X 0,Y 347.807,Z 607.157,A -85,B 0,C 180,E1 -13707.695,E2 -13707.695} C_VEL
LIN {X 0,Y 347.766,Z 607.161,A -85,B 0,C 180,E1 -13710.347,E2 -13710.347} C_VEL
LIN {X 0,Y 347.744,Z 607.164,A -85,B 0,C 180,E1 -13714.045,E2 -13714.045} C_VEL
LIN {X 0,Y 347.759,Z 607.164,A -85,B 0,C 180,E1 -13717.322,E2 -13717.322} C_VEL
LIN {X 0,Y 347.752,Z 607.164,A -85,B 0,C 180,E1 -13720.295,E2 -13720.295} C_VEL
LIN {X 0,Y 347.742,Z 607.167,A -85,B 0,C 180,E1 -13723.406,E2 -13723.406} C_VEL
LIN {X 0,Y 347.767,Z 607.166,A -85,B 0,C 180,E1 -13726.68,E2 -13726.68} C_VEL
LIN {X 0,Y 347.757,Z 607.166,A -85,B 0,C 180,E1 -13730.172,E2 -13730.172} C_VEL
LIN {X 0,Y 347.771,Z 607.169,A -85,B 0,C 180,E1 -13733.936,E2 -13733.936} C_VEL
LIN {X 0,Y 347.787,Z 607.273,A -85,B 0,C 180,E1 -13737.114,E2 -13737.114} C_VEL
LIN {X 0,Y 350.339,Z 617.805,A -85,B 0,C 180,E1 -13740.232,E2 -13740.232} C_VEL
LIN {X 0,Y 352.593,Z 628.931,A -85,B 0,C 180,E1 -13743.295,E2 -13743.295} C_VEL
LIN {X 0,Y 352.771,Z 631.731,A -85,B 0,C 180,E1 -13744.006,E2 -13744.006} C_VEL
LIN {X 0,Y 351.519,Z 641.62,A -85,B 0,C 180,E1 -13746.333,E2 -13746.333} C_VEL
LIN {X 0,Y 355.564,Z 663.194,A -85,B 0,C 180,E1 -13747.2,E2 -13747.2} C_VEL
LIN {X 0,Y 357.875,Z 680.434,A -85,B 0,C 180,E1 -13747.797,E2 -13747.797} C_VEL
LIN {X 0,Y 356.172,Z 750.975,A -85,B 0,C 180,E1 -13749.385,E2 -13749.385} C_VEL
LIN {X 0,Y 355.316,Z 764.495,A -85,B 0,C 180,E1 -13749.9,E2 -13749.9} C_VEL
LIN {X 0,Y 354.309,Z 776.871,A -85,B 0,C 180,E1 -13750.595,E2 -13750.595} C_VEL
LIN {X 0,Y 353.219,Z 788.037,A -85,B 0,C 180,E1 -13751.437,E2 -13751.437} C_VEL
LIN {X 0,Y 351.887,Z 799.687,A -85,B 0,C 180,E1 -13752.568,E2 -13752.568} C_VEL
LIN {X 0,Y 350.754,Z 809.144,A -85,B 0,C 180,E1 -13753.709,E2 -13753.709} C_VEL
LIN {X 0,Y 349.623,Z 818.873,A -85,B 0,C 180,E1 -13755.15,E2 -13755.15} C_VEL
LIN {X 0,Y 348.65,Z 826.897,A -85,B 0,C 180,E1 -13756.596,E2 -13756.596} C_VEL
LIN {X 0,Y 347.588,Z 834.748,A -85,B 0,C 180,E1 -13758.335,E2 -13758.335} C_VEL
LIN {X 0,Y 346.973,Z 841.078,A -85,B 0,C 180,E1 -13760.086,E2 -13760.086} C_VEL
LIN {X 0,Y 346.523,Z 846.122,A -85,B 0,C 180,E1 -13761.838,E2 -13761.838} C_VEL
LIN {X 0,Y 346.289,Z 850.025,A -85,B 0,C 180,E1 -13763.592,E2 -13763.592} C_VEL
LIN {X 0,Y 346.216,Z 852.888,A -85,B 0,C 180,E1 -13765.343,E2 -13765.343} C_VEL
LIN {X 0,Y 346.186,Z 854.251,A -85,B 0,C 180,E1 -13766.508,E2 -13766.508} C_VEL
LIN {X 0,Y 346.181,Z 855.213,A -85,B 0,C 180,E1 -13767.673,E2 -13767.673} C_VEL
LIN {X 0,Y 346.263,Z 855.736,A -85,B 0,C 180,E1 -13768.837,E2 -13768.837} C_VEL
LIN {X 0,Y 346.334,Z 855.838,A -85,B 0,C 180,E1 -13770,E2 -13770} C_VEL
LIN {X 0,Y 346.296,Z 855.536,A -85,B 0,C 180,E1 -13771.163,E2 -13771.163} C_VEL
LIN {X 0,Y 346.196,Z 854.83,A -85,B 0,C 180,E1 -13772.327,E2 -13772.327} C_VEL
LIN {X 0,Y 346.185,Z 853.675,A -85,B 0,C 180,E1 -13773.492,E2 -13773.492} C_VEL
LIN {X 0,Y 346.202,Z 851.143,A -85,B 0,C 180,E1 -13775.241,E2 -13775.241} C_VEL
LIN {X 0,Y 346.343,Z 847.565,A -85,B 0,C 180,E1 -13776.993,E2 -13776.993} C_VEL
LIN {X 0,Y 346.649,Z 842.844,A -85,B 0,C 180,E1 -13778.746,E2 -13778.746} C_VEL
LIN {X 0,Y 347.087,Z 836.834,A -85,B 0,C 180,E1 -13780.5,E2 -13780.5} C_VEL
LIN {X 0,Y 347.853,Z 829.335,A -85,B 0,C 180,E1 -13782.248,E2 -13782.248} C_VEL
LIN {X 0,Y 348.606,Z 821.678,A -85,B 0,C 180,E1 -13783.702,E2 -13783.702} C_VEL
LIN {X 0,Y 349.541,Z 812.209,A -85,B 0,C 180,E1 -13785.179,E2 -13785.179} C_VEL
LIN {X 0,Y 350.545,Z 802.071,A -85,B 0,C 180,E1 -13786.45,E2 -13786.45} C_VEL
LIN {X 0,Y 351.744,Z 790.656,A -85,B 0,C 180,E1 -13787.59,E2 -13787.59} C_VEL
LIN {X 0,Y 352.686,Z 778.809,A -85,B 0,C 180,E1 -13788.517,E2 -13788.517} C_VEL
LIN {X 0,Y 353.628,Z 765.846,A -85,B 0,C 180,E1 -13789.255,E2 -13789.255} C_VEL
LIN {X 0,Y 354.366,Z 752.203,A -85,B 0,C 180,E1 -13789.779,E2 -13789.779} C_VEL
LIN {X 0,Y 355.779,Z 679.732,A -85,B 0,C 180,E1 -13791.376,E2 -13791.376} C_VEL
LIN {X 0,Y 350.57,Z 643.47,A -85,B 0,C 180,E1 -13792.516,E2 -13792.516} C_VEL
LIN {X 0,Y 352.131,Z 629.444,A -85,B 0,C 180,E1 -13795.727,E2 -13795.727} C_VEL
LIN {X 0,Y 351.128,Z 622.663,A -85,B 0,C 180,E1 -13797.409,E2 -13797.409} C_VEL
LIN {X 0,Y 348.451,Z 610.311,A -85,B 0,C 180,E1 -13800.615,E2 -13800.615} C_VEL
LIN {X 0,Y 347.763,Z 607.167,A -85,B 0,C 180,E1 -13801.484,E2 -13801.484} C_VEL
LIN {X 0,Y 347.744,Z 607.171,A -85,B 0,C 180,E1 -13804.463,E2 -13804.463} C_VEL
LIN {X 0,Y 347.776,Z 607.162,A -85,B 0,C 180,E1 -13807.988,E2 -13807.988} C_VEL
LIN {X 0,Y 347.765,Z 607.162,A -85,B 0,C 180,E1 -13811.827,E2 -13811.827} C_VEL
LIN {X 0,Y 347.766,Z 607.165,A -85,B 0,C 180,E1 -13815.015,E2 -13815.015} C_VEL
LIN {X 0,Y 347.765,Z 607.165,A -85,B 0,C 180,E1 -13818.393,E2 -13818.393} C_VEL
LIN {X 0,Y 347.777,Z 607.161,A -85,B 0,C 180,E1 -13822.009,E2 -13822.009} C_VEL
LIN {X 0,Y 347.741,Z 607.166,A -85,B 0,C 180,E1 -13825.535,E2 -13825.535} C_VEL
LIN {X 0,Y 347.76,Z 607.164,A -85,B 0,C 180,E1 -13828.301,E2 -13828.301} C_VEL
LIN {X 0,Y 347.802,Z 607.163,A -85,B 0,C 180,E1 -13830.989,E2 -13830.989} C_VEL
LIN {X 0,Y 347.826,Z 607.155,A -85,B 0,C 180,E1 -13833.607,E2 -13833.607} C_VEL
LIN {X 0,Y 347.78,Z 607.16,A -85,B 0,C 180,E1 -13836.161,E2 -13836.161} C_VEL
LIN {X 0,Y 347.8,Z 607.158,A -85,B 0,C 180,E1 -13839.908,E2 -13839.908} C_VEL
LIN {X 0,Y 347.859,Z 607.151,A -85,B 0,C 180,E1 -13842.358,E2 -13842.358} C_VEL
LIN {X 0,Y 347.891,Z 607.147,A -85,B 0,C 180,E1 -13845.97,E2 -13845.97} C_VEL
LIN {X 0,Y 347.921,Z 607.146,A -85,B 0,C 180,E1 -13849.525,E2 -13849.525} C_VEL
LIN {X 0,Y 348.086,Z 607.126,A -85,B 0,C 180,E1 -13853.041,E2 -13853.041} C_VEL
LIN {X 0,Y 348.2,Z 607.111,A -85,B 0,C 180,E1 -13857.686,E2 -13857.686} C_VEL
LIN {X 0,Y 348.36,Z 607.089,A -85,B 0,C 180,E1 -13859.999,E2 -13859.999} C_VEL
LIN {X 0,Y 348.2,Z 607.108,A -85,B 0,C 180,E1 -13862.313,E2 -13862.313} C_VEL
LIN {X 0,Y 348.088,Z 607.123,A -85,B 0,C 180,E1 -13866.957,E2 -13866.957} C_VEL
LIN {X 0,Y 347.921,Z 607.143,A -85,B 0,C 180,E1 -13870.474,E2 -13870.474} C_VEL
LIN {X 0,Y 347.89,Z 607.149,A -85,B 0,C 180,E1 -13874.15,E2 -13874.15} C_VEL
LIN {X 0,Y 347.882,Z 607.149,A -85,B 0,C 180,E1 -13878.29,E2 -13878.29} C_VEL
LIN {X 0,Y 347.78,Z 607.164,A -85,B 0,C 180,E1 -13881.635,E2 -13881.635} C_VEL
LIN {X 0,Y 347.803,Z 607.158,A -85,B 0,C 180,E1 -13885.108,E2 -13885.108} C_VEL
LIN {X 0,Y 347.804,Z 607.161,A -85,B 0,C 180,E1 -13887.694,E2 -13887.694} C_VEL
LIN {X 0,Y 347.762,Z 607.165,A -85,B 0,C 180,E1 -13890.346,E2 -13890.346} C_VEL
LIN {X 0,Y 347.74,Z 607.172,A -85,B 0,C 180,E1 -13894.044,E2 -13894.044} C_VEL
LIN {X 0,Y 347.756,Z 607.163,A -85,B 0,C 180,E1 -13897.321,E2 -13897.321} C_VEL
LIN {X 0,Y 347.786,Z 607.165,A -85,B 0,C 180,E1 -13900.289,E2 -13900.289} C_VEL
LIN {X 0,Y 347.78,Z 607.16,A -85,B 0,C 180,E1 -13903.398,E2 -13903.398} C_VEL
LIN {X 0,Y 347.763,Z 607.165,A -85,B 0,C 180,E1 -13906.679,E2 -13906.679} C_VEL
LIN {X 0,Y 347.751,Z 607.168,A -85,B 0,C 180,E1 -13910.171,E2 -13910.171} C_VEL
LIN {X 0,Y 347.76,Z 607.166,A -85,B 0,C 180,E1 -13912.68,E2 -13912.68} C_VEL
LIN {X 0,Y 347.742,Z 607.167,A -85,B 0,C 180,E1 -13915.957,E2 -13915.957} C_VEL
LIN {X 0,Y 347.744,Z 607.165,A -85,B 0,C 180,E1 -13919.652,E2 -13919.652} C_VEL
LIN {X 0,Y 347.826,Z 607.154,A -85,B 0,C 180,E1 -13923.608,E2 -13923.608} C_VEL
LIN {X 0,Y 347.785,Z 607.161,A -85,B 0,C 180,E1 -13926.162,E2 -13926.162} C_VEL
LIN {X 0,Y 347.808,Z 607.157,A -85,B 0,C 180,E1 -13929.91,E2 -13929.91} C_VEL
LIN {X 0,Y 347.862,Z 607.152,A -85,B 0,C 180,E1 -13932.36,E2 -13932.36} C_VEL
LIN {X 0,Y 347.894,Z 607.146,A -85,B 0,C 180,E1 -13935.971,E2 -13935.971} C_VEL
LIN {X 0,Y 347.925,Z 607.143,A -85,B 0,C 180,E1 -13939.526,E2 -13939.526} C_VEL
LIN {X 0,Y 348.088,Z 607.127,A -85,B 0,C 180,E1 -13943.042,E2 -13943.042} C_VEL
LIN {X 0,Y 348.205,Z 607.108,A -85,B 0,C 180,E1 -13947.687,E2 -13947.687} C_VEL
LIN {X 0,Y 348.343,Z 607.09,A -85,B 0,C 180,E1 -13950,E2 -13950} C_VEL
LIN {X 0,Y 348.206,Z 607.107,A -85,B 0,C 180,E1 -13952.313,E2 -13952.313} C_VEL
LIN {X 0,Y 348.087,Z 607.126,A -85,B 0,C 180,E1 -13956.958,E2 -13956.958} C_VEL
LIN {X 0,Y 347.925,Z 607.142,A -85,B 0,C 180,E1 -13960.474,E2 -13960.474} C_VEL
LIN {X 0,Y 347.895,Z 607.146,A -85,B 0,C 180,E1 -13964.15,E2 -13964.15} C_VEL
LIN {X 0,Y 347.886,Z 607.151,A -85,B 0,C 180,E1 -13968.29,E2 -13968.29} C_VEL
LIN {X 0,Y 347.833,Z 607.273,A -85,B 0,C 180,E1 -13971.055,E2 -13971.055} C_VEL
LIN {X 0,Y 348.739,Z 611.862,A -85,B 0,C 180,E1 -13972.471,E2 -13972.471} C_VEL
LIN {X 0,Y 354.886,Z 629.729,A -85,B 0,C 180,E1 -13973.255,E2 -13973.255} C_VEL
LIN {X 0,Y 356.435,Z 637.763,A -85,B 0,C 180,E1 -13973.53,E2 -13973.53} C_VEL
LIN {X 0,Y 354.59,Z 718.783,A -85,B 0,C 180,E1 -13975.3,E2 -13975.3} C_VEL
LIN {X 0,Y 354.058,Z 732.815,A -85,B 0,C 180,E1 -13975.853,E2 -13975.853} C_VEL
LIN {X 0,Y 353.325,Z 745.601,A -85,B 0,C 180,E1 -13976.599,E2 -13976.599} C_VEL
LIN {X 0,Y 352.489,Z 756.589,A -85,B 0,C 180,E1 -13977.455,E2 -13977.455} C_VEL
LIN {X 0,Y 351.608,Z 767.297,A -85,B 0,C 180,E1 -13978.515,E2 -13978.515} C_VEL
LIN {X 0,Y 350.562,Z 777.379,A -85,B 0,C 180,E1 -13979.747,E2 -13979.747} C_VEL
LIN {X 0,Y 349.611,Z 787.036,A -85,B 0,C 180,E1 -13981.208,E2 -13981.208} C_VEL
LIN {X 0,Y 348.826,Z 794.398,A -85,B 0,C 180,E1 -13982.566,E2 -13982.566} C_VEL
LIN {X 0,Y 348.454,Z 797.459,A -85,B 0,C 180,E1 -13983.21,E2 -13983.21} C_VEL
LIN {X 0,Y 347.388,Z 800.975,A -85,B 0,C 180,E1 -13983.975,E2 -13983.975} C_VEL
LIN {X 0,Y 344.026,Z 806.217,A -85,B 0,C 180,E1 -13985.257,E2 -13985.257} C_VEL
LIN {X 0,Y 340.761,Z 810.729,A -85,B 0,C 180,E1 -13986.633,E2 -13986.633} C_VEL
LIN {X 0,Y 339.861,Z 813.101,A -85,B 0,C 180,E1 -13987.534,E2 -13987.534} C_VEL
LIN {X 0,Y 339.492,Z 816.67,A -85,B 0,C 180,E1 -13989.152,E2 -13989.152} C_VEL
LIN {X 0,Y 339.239,Z 819.326,A -85,B 0,C 180,E1 -13990.735,E2 -13990.735} C_VEL
LIN {X 0,Y 339.123,Z 820.61,A -85,B 0,C 180,E1 -13991.75,E2 -13991.75} C_VEL
LIN {X 0,Y 338.974,Z 822.089,A -85,B 0,C 180,E1 -13993.477,E2 -13993.477} C_VEL
LIN {X 0,Y 338.927,Z 822.692,A -85,B 0,C 180,E1 -13995.169,E2 -13995.169} C_VEL
LIN {X 0,Y 339.009,Z 822.496,A -85,B 0,C 180,E1 -13996.834,E2 -13996.834} C_VEL
LIN {X 0,Y 339.199,Z 821.545,A -85,B 0,C 180,E1 -13998.47,E2 -13998.47} C_VEL
LIN {X 0,Y 339.468,Z 819.846,A -85,B 0,C 180,E1 -14000.075,E2 -14000.075} C_VEL
LIN {X 0,Y 339.84,Z 817.141,A -85,B 0,C 180,E1 -14001.798,E2 -14001.798} C_VEL
LIN {X 0,Y 340.369,Z 813.208,A -85,B 0,C 180,E1 -14003.635,E2 -14003.635} C_VEL
LIN {X 0,Y 341.114,Z 807.978,A -85,B 0,C 180,E1 -14005.498,E2 -14005.498} C_VEL
LIN {X 0,Y 342.067,Z 801.136,A -85,B 0,C 180,E1 -14007.389,E2 -14007.389} C_VEL
LIN {X 0,Y 343.293,Z 792.781,A -85,B 0,C 180,E1 -14009.216,E2 -14009.216} C_VEL
LIN {X 0,Y 344.584,Z 783.477,A -85,B 0,C 180,E1 -14010.839,E2 -14010.839} C_VEL
LIN {X 0,Y 345.88,Z 773.242,A -85,B 0,C 180,E1 -14012.266,E2 -14012.266} C_VEL
LIN {X 0,Y 347.01,Z 763.236,A -85,B 0,C 180,E1 -14013.393,E2 -14013.393} C_VEL
LIN {X 0,Y 348.207,Z 751.445,A -85,B 0,C 180,E1 -14014.443,E2 -14014.443} C_VEL
LIN {X 0,Y 349.139,Z 739.551,A -85,B 0,C 180,E1 -14015.245,E2 -14015.245} C_VEL
LIN {X 0,Y 349.75,Z 726.908,A -85,B 0,C 180,E1 -14015.872,E2 -14015.872} C_VEL
LIN {X 0,Y 350.326,Z 713.913,A -85,B 0,C 180,E1 -14016.267,E2 -14016.267} C_VEL
LIN {X 0,Y 352.341,Z 639.539,A -85,B 0,C 180,E1 -14017.961,E2 -14017.961} C_VEL
LIN {X 0,Y 350.867,Z 634.479,A -85,B 0,C 180,E1 -14018.212,E2 -14018.212} C_VEL
LIN {X 0,Y 343.617,Z 617.614,A -85,B 0,C 180,E1 -14019.288,E2 -14019.288} C_VEL
LIN {X 0,Y 342.208,Z 614.356,A -85,B 0,C 180,E1 -14019.53,E2 -14019.53} C_VEL
LIN {X 0,Y 340.838,Z 608.031,A -85,B 0,C 180,E1 -14021.836,E2 -14021.836} C_VEL
LIN {X 0,Y 340.861,Z 608.027,A -85,B 0,C 180,E1 -14025.705,E2 -14025.705} C_VEL
LIN {X 0,Y 340.867,Z 608.028,A -85,B 0,C 180,E1 -14029.307,E2 -14029.307} C_VEL
LIN {X 0,Y 341.07,Z 608.002,A -85,B 0,C 180,E1 -14032.899,E2 -14032.899} C_VEL
LIN {X 0,Y 341.171,Z 607.987,A -85,B 0,C 180,E1 -14037.639,E2 -14037.639} C_VEL
LIN {X 0,Y 341.309,Z 607.969,A -85,B 0,C 180,E1 -14040.001,E2 -14040.001} C_VEL
LIN {X 0,Y 341.163,Z 607.987,A -85,B 0,C 180,E1 -14042.362,E2 -14042.362} C_VEL
LIN {X 0,Y 341.071,Z 607.997,A -85,B 0,C 180,E1 -14047.102,E2 -14047.102} C_VEL
LIN {X 0,Y 340.868,Z 608.022,A -85,B 0,C 180,E1 -14050.694,E2 -14050.694} C_VEL
LIN {X 0,Y 340.856,Z 608.025,A -85,B 0,C 180,E1 -14054.326,E2 -14054.326} C_VEL
LIN {X 0,Y 340.831,Z 608.029,A -85,B 0,C 180,E1 -14058.467,E2 -14058.467} C_VEL
LIN {X 0,Y 340.748,Z 608.035,A -85,B 0,C 180,E1 -14061.858,E2 -14061.858} C_VEL
LIN {X 0,Y 340.767,Z 608.03,A -85,B 0,C 180,E1 -14065.665,E2 -14065.665} C_VEL
LIN {X 0,Y 340.737,Z 608.036,A -85,B 0,C 180,E1 -14068.321,E2 -14068.321} C_VEL
LIN {X 0,Y 340.712,Z 608.042,A -85,B 0,C 180,E1 -14071.044,E2 -14071.044} C_VEL
LIN {X 0,Y 340.714,Z 608.038,A -85,B 0,C 180,E1 -14075.28,E2 -14075.28} C_VEL
LIN {X 0,Y 340.709,Z 608.039,A -85,B 0,C 180,E1 -14078.388,E2 -14078.388} C_VEL
LIN {X 0,Y 340.728,Z 608.043,A -85,B 0,C 180,E1 -14082.052,E2 -14082.052} C_VEL
LIN {X 0,Y 340.698,Z 608.045,A -85,B 0,C 180,E1 -14086.22,E2 -14086.22} C_VEL
LIN {X 0,Y 340.709,Z 608.045,A -85,B 0,C 180,E1 -14089.75,E2 -14089.75} C_VEL
LIN {X 0,Y 340.705,Z 608.046,A -85,B 0,C 180,E1 -14093.26,E2 -14093.26} C_VEL
LIN {X 0,Y 340.702,Z 608.056,A -85,B 0,C 180,E1 -14096.511,E2 -14096.511} C_VEL
LIN {X 0,Y 342.998,Z 617.39,A -85,B 0,C 180,E1 -14099.382,E2 -14099.382} C_VEL
LIN {X 0,Y 344.999,Z 626.685,A -85,B 0,C 180,E1 -14102.062,E2 -14102.062} C_VEL
LIN {X 0,Y 345.903,Z 631.747,A -85,B 0,C 180,E1 -14103.45,E2 -14103.45} C_VEL
LIN {X 0,Y 345.44,Z 636.844,A -85,B 0,C 180,E1 -14104.708,E2 -14104.708} C_VEL
LIN {X 0,Y 344.892,Z 641.105,A -85,B 0,C 180,E1 -14105.734,E2 -14105.734} C_VEL
LIN {X 0,Y 348.913,Z 662.528,A -85,B 0,C 180,E1 -14106.648,E2 -14106.648} C_VEL
LIN {X 0,Y 351.408,Z 680.805,A -85,B 0,C 180,E1 -14107.311,E2 -14107.311} C_VEL
LIN {X 0,Y 349.62,Z 751.17,A -85,B 0,C 180,E1 -14108.942,E2 -14108.942} C_VEL
LIN {X 0,Y 348.712,Z 765.233,A -85,B 0,C 180,E1 -14109.502,E2 -14109.502} C_VEL
LIN {X 0,Y 347.653,Z 777.285,A -85,B 0,C 180,E1 -14110.208,E2 -14110.208} C_VEL
LIN {X 0,Y 346.334,Z 789.835,A -85,B 0,C 180,E1 -14111.208,E2 -14111.208} C_VEL
LIN {X 0,Y 344.96,Z 801.102,A -85,B 0,C 180,E1 -14112.359,E2 -14112.359} C_VEL
LIN {X 0,Y 343.688,Z 811.299,A -85,B 0,C 180,E1 -14113.671,E2 -14113.671} C_VEL
LIN {X 0,Y 342.499,Z 820.53,A -85,B 0,C 180,E1 -14115.138,E2 -14115.138} C_VEL
LIN {X 0,Y 341.326,Z 829.567,A -85,B 0,C 180,E1 -14116.91,E2 -14116.91} C_VEL
LIN {X 0,Y 340.332,Z 836.851,A -85,B 0,C 180,E1 -14118.687,E2 -14118.687} C_VEL
LIN {X 0,Y 339.754,Z 842.686,A -85,B 0,C 180,E1 -14120.475,E2 -14120.475} C_VEL
LIN {X 0,Y 339.374,Z 847.308,A -85,B 0,C 180,E1 -14122.264,E2 -14122.264} C_VEL
LIN {X 0,Y 339.172,Z 850.832,A -85,B 0,C 180,E1 -14124.053,E2 -14124.053} C_VEL
LIN {X 0,Y 339.116,Z 852.596,A -85,B 0,C 180,E1 -14125.245,E2 -14125.245} C_VEL
LIN {X 0,Y 339.109,Z 853.949,A -85,B 0,C 180,E1 -14126.435,E2 -14126.435} C_VEL
LIN {X 0,Y 339.09,Z 854.895,A -85,B 0,C 180,E1 -14127.624,E2 -14127.624} C_VEL
LIN {X 0,Y 339.167,Z 855.393,A -85,B 0,C 180,E1 -14128.813,E2 -14128.813} C_VEL
LIN {X 0,Y 339.256,Z 855.483,A -85,B 0,C 180,E1 -14130,E2 -14130} C_VEL
LIN {X 0,Y 339.2,Z 855.166,A -85,B 0,C 180,E1 -14131.187,E2 -14131.187} C_VEL
LIN {X 0,Y 339.103,Z 854.442,A -85,B 0,C 180,E1 -14132.376,E2 -14132.376} C_VEL
LIN {X 0,Y 339.109,Z 853.26,A -85,B 0,C 180,E1 -14133.565,E2 -14133.565} C_VEL
LIN {X 0,Y 339.122,Z 850.48,A -85,B 0,C 180,E1 -14135.468,E2 -14135.468} C_VEL
LIN {X 0,Y 339.27,Z 847.077,A -85,B 0,C 180,E1 -14137.14,E2 -14137.14} C_VEL
LIN {X 0,Y 339.587,Z 842.314,A -85,B 0,C 180,E1 -14138.929,E2 -14138.929} C_VEL
LIN {X 0,Y 340.045,Z 836.257,A -85,B 0,C 180,E1 -14140.72,E2 -14140.72} C_VEL
LIN {X 0,Y 340.855,Z 828.706,A -85,B 0,C 180,E1 -14142.503,E2 -14142.503} C_VEL
LIN {X 0,Y 341.677,Z 820.99,A -85,B 0,C 180,E1 -14143.986,E2 -14143.986} C_VEL
LIN {X 0,Y 342.636,Z 811.615,A -85,B 0,C 180,E1 -14145.465,E2 -14145.465} C_VEL
LIN {X 0,Y 343.699,Z 801.174,A -85,B 0,C 180,E1 -14146.787,E2 -14146.787} C_VEL
LIN {X 0,Y 344.954,Z 789.637,A -85,B 0,C 180,E1 -14147.947,E2 -14147.947} C_VEL
LIN {X 0,Y 345.955,Z 777.545,A -85,B 0,C 180,E1 -14148.89,E2 -14148.89} C_VEL
LIN {X 0,Y 346.931,Z 764.23,A -85,B 0,C 180,E1 -14149.642,E2 -14149.642} C_VEL
LIN {X 0,Y 347.613,Z 751.052,A -85,B 0,C 180,E1 -14150.141,E2 -14150.141} C_VEL
LIN {X 0,Y 348.988,Z 679.95,A -85,B 0,C 180,E1 -14151.739,E2 -14151.739} C_VEL
LIN {X 0,Y 343.711,Z 643.15,A -85,B 0,C 180,E1 -14152.933,E2 -14152.933} C_VEL
LIN {X 0,Y 345.19,Z 630.504,A -85,B 0,C 180,E1 -14155.884,E2 -14155.884} C_VEL
LIN {X 0,Y 343.784,Z 622.015,A -85,B 0,C 180,E1 -14158.046,E2 -14158.046} C_VEL
LIN {X 0,Y 340.715,Z 608.046,A -85,B 0,C 180,E1 -14161.797,E2 -14161.797} C_VEL
LIN {X 0,Y 340.718,Z 608.04,A -85,B 0,C 180,E1 -14165.278,E2 -14165.278} C_VEL
LIN {X 0,Y 340.717,Z 608.045,A -85,B 0,C 180,E1 -14168.387,E2 -14168.387} C_VEL
LIN {X 0,Y 340.732,Z 608.04,A -85,B 0,C 180,E1 -14172.051,E2 -14172.051} C_VEL
LIN {X 0,Y 340.688,Z 608.044,A -85,B 0,C 180,E1 -14175.461,E2 -14175.461} C_VEL
LIN {X 0,Y 340.702,Z 608.048,A -85,B 0,C 180,E1 -14178.692,E2 -14178.692} C_VEL
LIN {X 0,Y 340.739,Z 608.037,A -85,B 0,C 180,E1 -14181.773,E2 -14181.773} C_VEL
LIN {X 0,Y 340.719,Z 608.04,A -85,B 0,C 180,E1 -14185.594,E2 -14185.594} C_VEL
LIN {X 0,Y 340.712,Z 608.047,A -85,B 0,C 180,E1 -14188.956,E2 -14188.956} C_VEL
LIN {X 0,Y 340.775,Z 608.035,A -85,B 0,C 180,E1 -14192.473,E2 -14192.473} C_VEL
LIN {X 0,Y 340.749,Z 608.037,A -85,B 0,C 180,E1 -14195.637,E2 -14195.637} C_VEL
LIN {X 0,Y 340.728,Z 608.041,A -85,B 0,C 180,E1 -14199.472,E2 -14199.472} C_VEL
LIN {X 0,Y 340.851,Z 608.023,A -85,B 0,C 180,E1 -14201.983,E2 -14201.983} C_VEL
LIN {X 0,Y 340.863,Z 608.023,A -85,B 0,C 180,E1 -14205.704,E2 -14205.704} C_VEL
LIN {X 0,Y 340.863,Z 608.028,A -85,B 0,C 180,E1 -14209.305,E2 -14209.305} C_VEL
LIN {X 0,Y 341.054,Z 608,A -85,B 0,C 180,E1 -14212.897,E2 -14212.897} C_VEL
LIN {X 0,Y 341.162,Z 607.989,A -85,B 0,C 180,E1 -14217.638,E2 -14217.638} C_VEL
LIN {X 0,Y 341.309,Z 607.968,A -85,B 0,C 180,E1 -14219.999,E2 -14219.999} C_VEL
LIN {X 0,Y 341.162,Z 607.985,A -85,B 0,C 180,E1 -14222.361,E2 -14222.361} C_VEL
LIN {X 0,Y 341.055,Z 608,A -85,B 0,C 180,E1 -14227.102,E2 -14227.102} C_VEL
LIN {X 0,Y 340.863,Z 608.022,A -85,B 0,C 180,E1 -14230.693,E2 -14230.693} C_VEL
LIN {X 0,Y 340.855,Z 608.024,A -85,B 0,C 180,E1 -14234.325,E2 -14234.325} C_VEL
LIN {X 0,Y 340.828,Z 608.027,A -85,B 0,C 180,E1 -14238.466,E2 -14238.466} C_VEL
LIN {X 0,Y 340.746,Z 608.043,A -85,B 0,C 180,E1 -14241.857,E2 -14241.857} C_VEL
LIN {X 0,Y 340.764,Z 608.038,A -85,B 0,C 180,E1 -14245.664,E2 -14245.664} C_VEL
LIN {X 0,Y 340.734,Z 608.041,A -85,B 0,C 180,E1 -14248.32,E2 -14248.32} C_VEL
LIN {X 0,Y 340.708,Z 608.041,A -85,B 0,C 180,E1 -14251.043,E2 -14251.043} C_VEL
LIN {X 0,Y 340.71,Z 608.041,A -85,B 0,C 180,E1 -14255.279,E2 -14255.279} C_VEL
LIN {X 0,Y 340.71,Z 608.045,A -85,B 0,C 180,E1 -14258.388,E2 -14258.388} C_VEL
LIN {X 0,Y 340.719,Z 608.04,A -85,B 0,C 180,E1 -14261.304,E2 -14261.304} C_VEL
LIN {X 0,Y 340.731,Z 608.042,A -85,B 0,C 180,E1 -14264.53,E2 -14264.53} C_VEL
LIN {X 0,Y 340.726,Z 608.042,A -85,B 0,C 180,E1 -14267.948,E2 -14267.948} C_VEL
LIN {X 0,Y 340.731,Z 608.039,A -85,B 0,C 180,E1 -14271.773,E2 -14271.773} C_VEL
LIN {X 0,Y 340.717,Z 608.04,A -85,B 0,C 180,E1 -14275.596,E2 -14275.596} C_VEL
LIN {X 0,Y 340.692,Z 608.045,A -85,B 0,C 180,E1 -14278.956,E2 -14278.956} C_VEL
LIN {X 0,Y 340.798,Z 608.032,A -85,B 0,C 180,E1 -14283.02,E2 -14283.02} C_VEL
LIN {X 0,Y 340.725,Z 608.043,A -85,B 0,C 180,E1 -14286.928,E2 -14286.928} C_VEL
LIN {X 0,Y 340.787,Z 608.038,A -85,B 0,C 180,E1 -14290.734,E2 -14290.734} C_VEL
LIN {X 0,Y 340.783,Z 608.034,A -85,B 0,C 180,E1 -14293.219,E2 -14293.219} C_VEL
LIN {X 0,Y 340.84,Z 608.031,A -85,B 0,C 180,E1 -14296.891,E2 -14296.891} C_VEL
LIN {X 0,Y 340.923,Z 608.017,A -85,B 0,C 180,E1 -14300.508,E2 -14300.508} C_VEL
LIN {X 0,Y 341.056,Z 608.004,A -85,B 0,C 180,E1 -14302.898,E2 -14302.898} C_VEL
LIN {X 0,Y 341.167,Z 607.985,A -85,B 0,C 180,E1 -14307.639,E2 -14307.639} C_VEL
LIN {X 0,Y 341.294,Z 607.968,A -85,B 0,C 180,E1 -14310,E2 -14310} C_VEL
LIN {X 0,Y 341.167,Z 607.984,A -85,B 0,C 180,E1 -14312.361,E2 -14312.361} C_VEL
LIN {X 0,Y 341.055,Z 608.003,A -85,B 0,C 180,E1 -14317.102,E2 -14317.102} C_VEL
LIN {X 0,Y 340.868,Z 608.022,A -85,B 0,C 180,E1 -14320.694,E2 -14320.694} C_VEL
LIN {X 0,Y 340.859,Z 608.022,A -85,B 0,C 180,E1 -14324.325,E2 -14324.325} C_VEL
LIN {X 0,Y 340.852,Z 608.027,A -85,B 0,C 180,E1 -14328.476,E2 -14328.476} C_VEL
LIN {X 0,Y 340.772,Z 608.109,A -85,B 0,C 180,E1 -14330.76,E2 -14330.76} C_VEL
LIN {X 0,Y 341.616,Z 612.302,A -85,B 0,C 180,E1 -14332.044,E2 -14332.044} C_VEL
LIN {X 0,Y 348.374,Z 631.687,A -85,B 0,C 180,E1 -14332.922,E2 -14332.922} C_VEL
LIN {X 0,Y 349.731,Z 638.63,A -85,B 0,C 180,E1 -14333.167,E2 -14333.167} C_VEL
LIN {X 0,Y 347.798,Z 719.416,A -85,B 0,C 180,E1 -14334.973,E2 -14334.973} C_VEL
LIN {X 0,Y 347.263,Z 733.222,A -85,B 0,C 180,E1 -14335.531,E2 -14335.531} C_VEL
LIN {X 0,Y 346.527,Z 745.495,A -85,B 0,C 180,E1 -14336.255,E2 -14336.255} C_VEL
LIN {X 0,Y 345.562,Z 758.022,A -85,B 0,C 180,E1 -14337.262,E2 -14337.262} C_VEL
LIN {X 0,Y 344.664,Z 768.07,A -85,B 0,C 180,E1 -14338.289,E2 -14338.289} C_VEL
LIN {X 0,Y 343.586,Z 778.25,A -85,B 0,C 180,E1 -14339.568,E2 -14339.568} C_VEL
LIN {X 0,Y 342.65,Z 787.559,A -85,B 0,C 180,E1 -14341.019,E2 -14341.019} C_VEL
LIN {X 0,Y 341.626,Z 796.625,A -85,B 0,C 180,E1 -14342.775,E2 -14342.775} C_VEL
LIN {X 0,Y 340.836,Z 803.546,A -85,B 0,C 180,E1 -14344.434,E2 -14344.434} C_VEL
LIN {X 0,Y 340.205,Z 809.864,A -85,B 0,C 180,E1 -14346.326,E2 -14346.326} C_VEL
LIN {X 0,Y 339.861,Z 813.101,A -85,B 0,C 180,E1 -14347.534,E2 -14347.534} C_VEL
LIN {X 0,Y 338.973,Z 815.297,A -85,B 0,C 180,E1 -14348.453,E2 -14348.453} C_VEL
LIN {X 0,Y 335.809,Z 818.344,A -85,B 0,C 180,E1 -14349.964,E2 -14349.964} C_VEL
LIN {X 0,Y 333.21,Z 820.259,A -85,B 0,C 180,E1 -14351.212,E2 -14351.212} C_VEL
LIN {X 0,Y 332.071,Z 821.401,A -85,B 0,C 180,E1 -14352.195,E2 -14352.195} C_VEL
LIN {X 0,Y 331.962,Z 821.72,A -85,B 0,C 180,E1 -14352.53,E2 -14352.53} C_VEL
LIN {X 0,Y 331.847,Z 822.828,A -85,B 0,C 180,E1 -14354.337,E2 -14354.337} C_VEL
LIN {X 0,Y 331.866,Z 823.046,A -85,B 0,C 180,E1 -14356.055,E2 -14356.055} C_VEL
LIN {X 0,Y 332.012,Z 822.447,A -85,B 0,C 180,E1 -14357.805,E2 -14357.805} C_VEL
LIN {X 0,Y 332.282,Z 820.969,A -85,B 0,C 180,E1 -14359.588,E2 -14359.588} C_VEL
LIN {X 0,Y 332.689,Z 818.525,A -85,B 0,C 180,E1 -14361.407,E2 -14361.407} C_VEL
LIN {X 0,Y 333.166,Z 814.955,A -85,B 0,C 180,E1 -14363.281,E2 -14363.281} C_VEL
LIN {X 0,Y 334.002,Z 809.518,A -85,B 0,C 180,E1 -14365.381,E2 -14365.381} C_VEL
LIN {X 0,Y 335.04,Z 802.59,A -85,B 0,C 180,E1 -14367.434,E2 -14367.434} C_VEL
LIN {X 0,Y 336.253,Z 794.687,A -85,B 0,C 180,E1 -14369.254,E2 -14369.254} C_VEL
LIN {X 0,Y 337.633,Z 785.473,A -85,B 0,C 180,E1 -14370.954,E2 -14370.954} C_VEL
LIN {X 0,Y 338.881,Z 776.132,A -85,B 0,C 180,E1 -14372.353,E2 -14372.353} C_VEL
LIN {X 0,Y 340.187,Z 765.48,A -85,B 0,C 180,E1 -14373.63,E2 -14373.63} C_VEL
LIN {X 0,Y 341.52,Z 753.465,A -85,B 0,C 180,E1 -14374.761,E2 -14374.761} C_VEL
LIN {X 0,Y 342.544,Z 741.296,A -85,B 0,C 180,E1 -14375.636,E2 -14375.636} C_VEL
LIN {X 0,Y 343.237,Z 728.27,A -85,B 0,C 180,E1 -14376.313,E2 -14376.313} C_VEL
LIN {X 0,Y 343.817,Z 715.576,A -85,B 0,C 180,E1 -14376.727,E2 -14376.727} C_VEL
LIN {X 0,Y 345.915,Z 640.364,A -85,B 0,C 180,E1 -14378.48,E2 -14378.48} C_VEL
LIN {X 0,Y 341.902,Z 629.954,A -85,B 0,C 180,E1 -14379.115,E2 -14379.115} C_VEL
LIN {X 0,Y 335.076,Z 614.838,A -85,B 0,C 180,E1 -14380.193,E2 -14380.193} C_VEL
LIN {X 0,Y 333.757,Z 608.913,A -85,B 0,C 180,E1 -14382.46,E2 -14382.46} C_VEL
LIN {X 0,Y 333.8,Z 608.907,A -85,B 0,C 180,E1 -14385.577,E2 -14385.577} C_VEL
LIN {X 0,Y 333.83,Z 608.903,A -85,B 0,C 180,E1 -14389.079,E2 -14389.079} C_VEL
LIN {X 0,Y 334.019,Z 608.879,A -85,B 0,C 180,E1 -14392.748,E2 -14392.748} C_VEL
LIN {X 0,Y 334.133,Z 608.864,A -85,B 0,C 180,E1 -14397.59,E2 -14397.59} C_VEL
LIN {X 0,Y 334.259,Z 608.848,A -85,B 0,C 180,E1 -14400.001,E2 -14400.001} C_VEL
LIN {X 0,Y 334.124,Z 608.865,A -85,B 0,C 180,E1 -14402.412,E2 -14402.412} C_VEL
LIN {X 0,Y 334.02,Z 608.876,A -85,B 0,C 180,E1 -14407.253,E2 -14407.253} C_VEL
LIN {X 0,Y 333.831,Z 608.901,A -85,B 0,C 180,E1 -14410.923,E2 -14410.923} C_VEL
LIN {X 0,Y 333.802,Z 608.906,A -85,B 0,C 180,E1 -14414.635,E2 -14414.635} C_VEL
LIN {X 0,Y 333.79,Z 608.905,A -85,B 0,C 180,E1 -14418.656,E2 -14418.656} C_VEL
LIN {X 0,Y 333.687,Z 608.914,A -85,B 0,C 180,E1 -14422.279,E2 -14422.279} C_VEL
LIN {X 0,Y 333.731,Z 608.907,A -85,B 0,C 180,E1 -14426.247,E2 -14426.247} C_VEL
LIN {X 0,Y 333.707,Z 608.909,A -85,B 0,C 180,E1 -14428.973,E2 -14428.973} C_VEL
LIN {X 0,Y 333.647,Z 608.916,A -85,B 0,C 180,E1 -14432.59,E2 -14432.59} C_VEL
LIN {X 0,Y 333.673,Z 608.919,A -85,B 0,C 180,E1 -14436.14,E2 -14436.14} C_VEL
LIN {X 0,Y 333.667,Z 608.921,A -85,B 0,C 180,E1 -14439.19,E2 -14439.19} C_VEL
LIN {X 0,Y 333.664,Z 608.922,A -85,B 0,C 180,E1 -14442.507,E2 -14442.507} C_VEL
LIN {X 0,Y 333.645,Z 608.923,A -85,B 0,C 180,E1 -14445.965,E2 -14445.965} C_VEL
LIN {X 0,Y 333.655,Z 608.926,A -85,B 0,C 180,E1 -14449.315,E2 -14449.315} C_VEL
LIN {X 0,Y 333.655,Z 608.925,A -85,B 0,C 180,E1 -14452.35,E2 -14452.35} C_VEL
LIN {X 0,Y 333.681,Z 608.935,A -85,B 0,C 180,E1 -14455.891,E2 -14455.891} C_VEL
LIN {X 0,Y 336.298,Z 619.61,A -85,B 0,C 180,E1 -14459.287,E2 -14459.287} C_VEL
LIN {X 0,Y 338.345,Z 629.278,A -85,B 0,C 180,E1 -14462.137,E2 -14462.137} C_VEL
LIN {X 0,Y 339.076,Z 634.628,A -85,B 0,C 180,E1 -14463.612,E2 -14463.612} C_VEL
LIN {X 0,Y 338.249,Z 641.072,A -85,B 0,C 180,E1 -14465.152,E2 -14465.152} C_VEL
LIN {X 0,Y 342.301,Z 662.095,A -85,B 0,C 180,E1 -14466.079,E2 -14466.079} C_VEL
LIN {X 0,Y 345.001,Z 681.68,A -85,B 0,C 180,E1 -14466.815,E2 -14466.815} C_VEL
LIN {X 0,Y 343.163,Z 750.587,A -85,B 0,C 180,E1 -14468.448,E2 -14468.448} C_VEL
LIN {X 0,Y 342.179,Z 764.66,A -85,B 0,C 180,E1 -14469.014,E2 -14469.014} C_VEL
LIN {X 0,Y 341.115,Z 776.73,A -85,B 0,C 180,E1 -14469.734,E2 -14469.734} C_VEL
LIN {X 0,Y 339.822,Z 788.497,A -85,B 0,C 180,E1 -14470.677,E2 -14470.677} C_VEL
LIN {X 0,Y 338.384,Z 799.918,A -85,B 0,C 180,E1 -14471.848,E2 -14471.848} C_VEL
LIN {X 0,Y 336.956,Z 810.401,A -85,B 0,C 180,E1 -14473.194,E2 -14473.194} C_VEL
LIN {X 0,Y 335.624,Z 820.548,A -85,B 0,C 180,E1 -14474.84,E2 -14474.84} C_VEL
LIN {X 0,Y 334.398,Z 829.471,A -85,B 0,C 180,E1 -14476.633,E2 -14476.633} C_VEL
LIN {X 0,Y 333.341,Z 836.694,A -85,B 0,C 180,E1 -14478.446,E2 -14478.446} C_VEL
LIN {X 0,Y 332.731,Z 842.488,A -85,B 0,C 180,E1 -14480.272,E2 -14480.272} C_VEL
LIN {X 0,Y 332.31,Z 847.068,A -85,B 0,C 180,E1 -14482.099,E2 -14482.099} C_VEL
LIN {X 0,Y 332.094,Z 850.786,A -85,B 0,C 180,E1 -14484.074,E2 -14484.074} C_VEL
LIN {X 0,Y 332.033,Z 853.648,A -85,B 0,C 180,E1 -14486.359,E2 -14486.359} C_VEL
LIN {X 0,Y 332.001,Z 854.573,A -85,B 0,C 180,E1 -14487.574,E2 -14487.574} C_VEL
LIN {X 0,Y 332.07,Z 855.051,A -85,B 0,C 180,E1 -14488.787,E2 -14488.787} C_VEL
LIN {X 0,Y 332.164,Z 855.128,A -85,B 0,C 180,E1 -14490,E2 -14490} C_VEL
LIN {X 0,Y 332.103,Z 854.797,A -85,B 0,C 180,E1 -14491.213,E2 -14491.213} C_VEL
LIN {X 0,Y 332.013,Z 854.049,A -85,B 0,C 180,E1 -14492.426,E2 -14492.426} C_VEL
LIN {X 0,Y 332.034,Z 852.845,A -85,B 0,C 180,E1 -14493.641,E2 -14493.641} C_VEL
LIN {X 0,Y 332.092,Z 849.431,A -85,B 0,C 180,E1 -14495.923,E2 -14495.923} C_VEL
LIN {X 0,Y 332.309,Z 845.139,A -85,B 0,C 180,E1 -14497.901,E2 -14497.901} C_VEL
LIN {X 0,Y 332.764,Z 838.907,A -85,B 0,C 180,E1 -14500.034,E2 -14500.034} C_VEL
LIN {X 0,Y 333.4,Z 832.082,A -85,B 0,C 180,E1 -14501.86,E2 -14501.86} C_VEL
LIN {X 0,Y 334.364,Z 823.601,A -85,B 0,C 180,E1 -14503.678,E2 -14503.678} C_VEL
LIN {X 0,Y 335.3,Z 814.584,A -85,B 0,C 180,E1 -14505.228,E2 -14505.228} C_VEL
LIN {X 0,Y 336.41,Z 804.039,A -85,B 0,C 180,E1 -14506.693,E2 -14506.693} C_VEL
LIN {X 0,Y 337.619,Z 793.341,A -85,B 0,C 180,E1 -14507.881,E2 -14507.881} C_VEL
LIN {X 0,Y 338.79,Z 781.399,A -85,B 0,C 180,E1 -14508.912,E2 -14508.912} C_VEL
LIN {X 0,Y 339.808,Z 769.06,A -85,B 0,C 180,E1 -14509.717,E2 -14509.717} C_VEL
LIN {X 0,Y 340.593,Z 756.516,A -85,B 0,C 180,E1 -14510.298,E2 -14510.298} C_VEL
LIN {X 0,Y 341.109,Z 741.147,A -85,B 0,C 180,E1 -14510.724,E2 -14510.724} C_VEL
LIN {X 0,Y 342.292,Z 680.893,A -85,B 0,C 180,E1 -14512.095,E2 -14512.095} C_VEL
LIN {X 0,Y 336.832,Z 642.845,A -85,B 0,C 180,E1 -14513.355,E2 -14513.355} C_VEL
LIN {X 0,Y 338.173,Z 630.841,A -85,B 0,C 180,E1 -14516.227,E2 -14516.227} C_VEL
LIN {X 0,Y 336.363,Z 621.361,A -85,B 0,C 180,E1 -14518.721,E2 -14518.721} C_VEL
LIN {X 0,Y 333.657,Z 608.925,A -85,B 0,C 180,E1 -14522.159,E2 -14522.159} C_VEL
LIN {X 0,Y 333.676,Z 608.92,A -85,B 0,C 180,E1 -14526.138,E2 -14526.138} C_VEL
LIN {X 0,Y 333.671,Z 608.919,A -85,B 0,C 180,E1 -14529.188,E2 -14529.188} C_VEL
LIN {X 0,Y 333.674,Z 608.923,A -85,B 0,C 180,E1 -14532.507,E2 -14532.507} C_VEL
LIN {X 0,Y 333.631,Z 608.923,A -85,B 0,C 180,E1 -14535.96,E2 -14535.96} C_VEL
LIN {X 0,Y 333.654,Z 608.921,A -85,B 0,C 180,E1 -14539.312,E2 -14539.312} C_VEL
LIN {X 0,Y 333.655,Z 608.922,A -85,B 0,C 180,E1 -14542.349,E2 -14542.349} C_VEL
LIN {X 0,Y 333.671,Z 608.919,A -85,B 0,C 180,E1 -14545.34,E2 -14545.34} C_VEL
LIN {X 0,Y 333.696,Z 608.915,A -85,B 0,C 180,E1 -14549.637,E2 -14549.637} C_VEL
LIN {X 0,Y 333.74,Z 608.911,A -85,B 0,C 180,E1 -14552.4,E2 -14552.4} C_VEL
LIN {X 0,Y 333.721,Z 608.917,A -85,B 0,C 180,E1 -14555.09,E2 -14555.09} C_VEL
LIN {X 0,Y 333.668,Z 608.924,A -85,B 0,C 180,E1 -14559.018,E2 -14559.018} C_VEL
LIN {X 0,Y 333.787,Z 608.905,A -85,B 0,C 180,E1 -14561.588,E2 -14561.588} C_VEL
LIN {X 0,Y 333.802,Z 608.904,A -85,B 0,C 180,E1 -14565.576,E2 -14565.576} C_VEL
LIN {X 0,Y 333.826,Z 608.903,A -85,B 0,C 180,E1 -14569.077,E2 -14569.077} C_VEL
LIN {X 0,Y 334.006,Z 608.877,A -85,B 0,C 180,E1 -14572.746,E2 -14572.746} C_VEL
LIN {X 0,Y 333.806,Z 608.905,A -85,B 0,C 180,E1 -14575.168,E2 -14575.168} C_VEL
LIN {X 0,Y 334.1,Z 608.869,A -85,B 0,C 180,E1 -14577.588,E2 -14577.588} C_VEL
LIN {X 0,Y 334.259,Z 608.846,A -85,B 0,C 180,E1 -14579.999,E2 -14579.999} C_VEL
LIN {X 0,Y 334.1,Z 608.864,A -85,B 0,C 180,E1 -14582.411,E2 -14582.411} C_VEL
LIN {X 0,Y 333.99,Z 608.878,A -85,B 0,C 180,E1 -14586.632,E2 -14586.632} C_VEL
LIN {X 0,Y 333.853,Z 608.901,A -85,B 0,C 180,E1 -14589.695,E2 -14589.695} C_VEL
LIN {X 0,Y 333.788,Z 608.906,A -85,B 0,C 180,E1 -14593.391,E2 -14593.391} C_VEL
LIN {X 0,Y 333.737,Z 608.911,A -85,B 0,C 180,E1 -14597.146,E2 -14597.146} C_VEL
LIN {X 0,Y 333.727,Z 608.916,A -85,B 0,C 180,E1 -14599.69,E2 -14599.69} C_VEL
LIN {X 0,Y 333.684,Z 608.918,A -85,B 0,C 180,E1 -14602.278,E2 -14602.278} C_VEL
LIN {X 0,Y 333.727,Z 608.914,A -85,B 0,C 180,E1 -14606.246,E2 -14606.246} C_VEL
LIN {X 0,Y 333.704,Z 608.914,A -85,B 0,C 180,E1 -14608.972,E2 -14608.972} C_VEL
LIN {X 0,Y 333.643,Z 608.923,A -85,B 0,C 180,E1 -14612.589,E2 -14612.589} C_VEL
LIN {X 0,Y 333.669,Z 608.924,A -85,B 0,C 180,E1 -14616.139,E2 -14616.139} C_VEL
LIN {X 0,Y 333.677,Z 608.917,A -85,B 0,C 180,E1 -14619.187,E2 -14619.187} C_VEL
LIN {X 0,Y 333.684,Z 608.919,A -85,B 0,C 180,E1 -14622.511,E2 -14622.511} C_VEL
LIN {X 0,Y 333.653,Z 608.923,A -85,B 0,C 180,E1 -14625.966,E2 -14625.966} C_VEL
LIN {X 0,Y 333.65,Z 608.92,A -85,B 0,C 180,E1 -14629.314,E2 -14629.314} C_VEL
LIN {X 0,Y 333.649,Z 608.926,A -85,B 0,C 180,E1 -14632.35,E2 -14632.35} C_VEL
LIN {X 0,Y 333.668,Z 608.918,A -85,B 0,C 180,E1 -14635.342,E2 -14635.342} C_VEL
LIN {X 0,Y 333.685,Z 608.916,A -85,B 0,C 180,E1 -14639.637,E2 -14639.637} C_VEL
LIN {X 0,Y 333.734,Z 608.914,A -85,B 0,C 180,E1 -14642.401,E2 -14642.401} C_VEL
LIN {X 0,Y 333.722,Z 608.913,A -85,B 0,C 180,E1 -14645.091,E2 -14645.091} C_VEL
LIN {X 0,Y 333.681,Z 608.92,A -85,B 0,C 180,E1 -14649.02,E2 -14649.02} C_VEL
LIN {X 0,Y 333.789,Z 608.903,A -85,B 0,C 180,E1 -14651.59,E2 -14651.59} C_VEL
LIN {X 0,Y 333.805,Z 608.902,A -85,B 0,C 180,E1 -14655.577,E2 -14655.577} C_VEL
LIN {X 0,Y 333.83,Z 608.902,A -85,B 0,C 180,E1 -14659.078,E2 -14659.078} C_VEL
LIN {X 0,Y 334.009,Z 608.88,A -85,B 0,C 180,E1 -14662.747,E2 -14662.747} C_VEL
LIN {X 0,Y 333.807,Z 608.905,A -85,B 0,C 180,E1 -14665.169,E2 -14665.169} C_VEL
LIN {X 0,Y 334.104,Z 608.865,A -85,B 0,C 180,E1 -14667.589,E2 -14667.589} C_VEL
LIN {X 0,Y 334.244,Z 608.846,A -85,B 0,C 180,E1 -14670,E2 -14670} C_VEL
LIN {X 0,Y 334.105,Z 608.864,A -85,B 0,C 180,E1 -14672.411,E2 -14672.411} C_VEL
LIN {X 0,Y 334.011,Z 608.876,A -85,B 0,C 180,E1 -14676.039,E2 -14676.039} C_VEL
LIN {X 0,Y 333.955,Z 608.883,A -85,B 0,C 180,E1 -14678.471,E2 -14678.471} C_VEL
LIN {X 0,Y 333.788,Z 608.903,A -85,B 0,C 180,E1 -14682.154,E2 -14682.154} C_VEL
LIN {X 0,Y 333.774,Z 608.906,A -85,B 0,C 180,E1 -14685.886,E2 -14685.886} C_VEL
LIN {X 0,Y 333.801,Z 608.905,A -85,B 0,C 180,E1 -14688.659,E2 -14688.659} C_VEL
LIN {X 0,Y 333.733,Z 609.076,A -85,B 0,C 180,E1 -14690.493,E2 -14690.493} C_VEL
LIN {X 0,Y 334.415,Z 612.435,A -85,B 0,C 180,E1 -14691.578,E2 -14691.578} C_VEL
LIN {X 0,Y 341.937,Z 633.849,A -85,B 0,C 180,E1 -14692.587,E2 -14692.587} C_VEL
LIN {X 0,Y 343.037,Z 639.534,A -85,B 0,C 180,E1 -14692.79,E2 -14692.79} C_VEL
LIN {X 0,Y 341.037,Z 719.463,A -85,B 0,C 180,E1 -14694.613,E2 -14694.613} C_VEL
LIN {X 0,Y 340.482,Z 733.231,A -85,B 0,C 180,E1 -14695.176,E2 -14695.176} C_VEL
LIN {X 0,Y 339.74,Z 745.553,A -85,B 0,C 180,E1 -14695.912,E2 -14695.912} C_VEL
LIN {X 0,Y 338.776,Z 757.44,A -85,B 0,C 180,E1 -14696.87,E2 -14696.87} C_VEL
LIN {X 0,Y 337.717,Z 769.14,A -85,B 0,C 180,E1 -14698.088,E2 -14698.088} C_VEL
LIN {X 0,Y 336.603,Z 779.497,A -85,B 0,C 180,E1 -14699.439,E2 -14699.439} C_VEL
LIN {X 0,Y 335.657,Z 788.278,A -85,B 0,C 180,E1 -14700.857,E2 -14700.857} C_VEL
LIN {X 0,Y 334.632,Z 797.012,A -85,B 0,C 180,E1 -14702.589,E2 -14702.589} C_VEL
LIN {X 0,Y 333.834,Z 803.893,A -85,B 0,C 180,E1 -14704.273,E2 -14704.273} C_VEL
LIN {X 0,Y 333.149,Z 810.212,A -85,B 0,C 180,E1 -14706.204,E2 -14706.204} C_VEL
LIN {X 0,Y 332.722,Z 814.261,A -85,B 0,C 180,E1 -14707.774,E2 -14707.774} C_VEL
LIN {X 0,Y 332.373,Z 817.528,A -85,B 0,C 180,E1 -14709.37,E2 -14709.37} C_VEL
LIN {X 0,Y 332.107,Z 820.05,A -85,B 0,C 180,E1 -14710.996,E2 -14710.996} C_VEL
LIN {X 0,Y 331.962,Z 821.72,A -85,B 0,C 180,E1 -14712.53,E2 -14712.53} C_VEL
LIN {X 0,Y 331.23,Z 822.536,A -85,B 0,C 180,E1 -14713.533,E2 -14713.533} C_VEL
LIN {X 0,Y 328.31,Z 823.256,A -85,B 0,C 180,E1 -14715.175,E2 -14715.175} C_VEL
LIN {X 0,Y 325.921,Z 823.308,A -85,B 0,C 180,E1 -14716.51,E2 -14716.51} C_VEL
LIN {X 0,Y 324.971,Z 823.021,A -85,B 0,C 180,E1 -14717.542,E2 -14717.542} C_VEL
LIN {X 0,Y 324.932,Z 822.826,A -85,B 0,C 180,E1 -14717.891,E2 -14717.891} C_VEL
LIN {X 0,Y 325.194,Z 821.516,A -85,B 0,C 180,E1 -14719.584,E2 -14719.584} C_VEL
LIN {X 0,Y 325.591,Z 819.426,A -85,B 0,C 180,E1 -14721.247,E2 -14721.247} C_VEL
LIN {X 0,Y 326.233,Z 814.942,A -85,B 0,C 180,E1 -14723.687,E2 -14723.687} C_VEL
LIN {X 0,Y 326.955,Z 810.52,A -85,B 0,C 180,E1 -14725.445,E2 -14725.445} C_VEL
LIN {X 0,Y 328.075,Z 803.474,A -85,B 0,C 180,E1 -14727.62,E2 -14727.62} C_VEL
LIN {X 0,Y 329.098,Z 797.161,A -85,B 0,C 180,E1 -14729.168,E2 -14729.168} C_VEL
LIN {X 0,Y 330.502,Z 788.894,A -85,B 0,C 180,E1 -14730.827,E2 -14730.827} C_VEL
LIN {X 0,Y 331.838,Z 779.392,A -85,B 0,C 180,E1 -14732.37,E2 -14732.37} C_VEL
LIN {X 0,Y 333.235,Z 769.111,A -85,B 0,C 180,E1 -14733.712,E2 -14733.712} C_VEL
LIN {X 0,Y 334.458,Z 758.765,A -85,B 0,C 180,E1 -14734.799,E2 -14734.799} C_VEL
LIN {X 0,Y 335.604,Z 747.456,A -85,B 0,C 180,E1 -14735.735,E2 -14735.735} C_VEL
LIN {X 0,Y 336.549,Z 734.281,A -85,B 0,C 180,E1 -14736.543,E2 -14736.543} C_VEL
LIN {X 0,Y 337.191,Z 721.283,A -85,B 0,C 180,E1 -14737.087,E2 -14737.087} C_VEL
LIN {X 0,Y 339.624,Z 641.756,A -85,B 0,C 180,E1 -14739.008,E2 -14739.008} C_VEL
LIN {X 0,Y 333.143,Z 626.284,A -85,B 0,C 180,E1 -14740.05,E2 -14740.05} C_VEL
LIN {X 0,Y 327.984,Z 615.335,A -85,B 0,C 180,E1 -14740.899,E2 -14740.899} C_VEL
LIN {X 0,Y 326.693,Z 609.789,A -85,B 0,C 180,E1 -14743.118,E2 -14743.118} C_VEL
LIN {X 0,Y 326.752,Z 609.784,A -85,B 0,C 180,E1 -14746.315,E2 -14746.315} C_VEL
LIN {X 0,Y 326.808,Z 609.779,A -85,B 0,C 180,E1 -14750.094,E2 -14750.094} C_VEL
LIN {X 0,Y 326.973,Z 609.757,A -85,B 0,C 180,E1 -14752.591,E2 -14752.591} C_VEL
LIN {X 0,Y 326.78,Z 609.782,A -85,B 0,C 180,E1 -14755.066,E2 -14755.066} C_VEL
LIN {X 0,Y 327.07,Z 609.744,A -85,B 0,C 180,E1 -14757.538,E2 -14757.538} C_VEL
LIN {X 0,Y 327.21,Z 609.726,A -85,B 0,C 180,E1 -14760.001,E2 -14760.001} C_VEL
LIN {X 0,Y 327.061,Z 609.745,A -85,B 0,C 180,E1 -14762.464,E2 -14762.464} C_VEL
LIN {X 0,Y 326.992,Z 609.752,A -85,B 0,C 180,E1 -14766.17,E2 -14766.17} C_VEL
LIN {X 0,Y 326.908,Z 609.766,A -85,B 0,C 180,E1 -14768.656,E2 -14768.656} C_VEL
LIN {X 0,Y 326.732,Z 609.783,A -85,B 0,C 180,E1 -14772.422,E2 -14772.422} C_VEL
LIN {X 0,Y 326.748,Z 609.783,A -85,B 0,C 180,E1 -14774.958,E2 -14774.958} C_VEL
LIN {X 0,Y 326.727,Z 609.783,A -85,B 0,C 180,E1 -14778.839,E2 -14778.839} C_VEL
LIN {X 0,Y 326.615,Z 609.794,A -85,B 0,C 180,E1 -14782.788,E2 -14782.788} C_VEL
LIN {X 0,Y 326.685,Z 609.785,A -85,B 0,C 180,E1 -14785.485,E2 -14785.485} C_VEL
LIN {X 0,Y 326.657,Z 609.79,A -85,B 0,C 180,E1 -14789.66,E2 -14789.66} C_VEL
LIN {X 0,Y 326.619,Z 609.793,A -85,B 0,C 180,E1 -14792.949,E2 -14792.949} C_VEL
LIN {X 0,Y 326.628,Z 609.798,A -85,B 0,C 180,E1 -14797.048,E2 -14797.048} C_VEL
LIN {X 0,Y 326.601,Z 609.799,A -85,B 0,C 180,E1 -14800.208,E2 -14800.208} C_VEL
LIN {X 0,Y 326.59,Z 609.801,A -85,B 0,C 180,E1 -14803.522,E2 -14803.522} C_VEL
LIN {X 0,Y 326.612,Z 609.803,A -85,B 0,C 180,E1 -14807.022,E2 -14807.022} C_VEL
LIN {X 0,Y 326.642,Z 609.798,A -85,B 0,C 180,E1 -14811.395,E2 -14811.395} C_VEL
LIN {X 0,Y 326.654,Z 609.805,A -85,B 0,C 180,E1 -14815.24,E2 -14815.24} C_VEL
LIN {X 0,Y 329.179,Z 620.127,A -85,B 0,C 180,E1 -14818.651,E2 -14818.651} C_VEL
LIN {X 0,Y 331.204,Z 629.38,A -85,B 0,C 180,E1 -14821.483,E2 -14821.483} C_VEL
LIN {X 0,Y 332.262,Z 635.729,A -85,B 0,C 180,E1 -14823.309,E2 -14823.309} C_VEL
LIN {X 0,Y 331.606,Z 640.342,A -85,B 0,C 180,E1 -14824.481,E2 -14824.481} C_VEL
LIN {X 0,Y 335.991,Z 662.973,A -85,B 0,C 180,E1 -14825.536,E2 -14825.536} C_VEL
LIN {X 0,Y 338.673,Z 683.189,A -85,B 0,C 180,E1 -14826.322,E2 -14826.322} C_VEL
LIN {X 0,Y 336.746,Z 750.107,A -85,B 0,C 180,E1 -14827.935,E2 -14827.935} C_VEL
LIN {X 0,Y 335.746,Z 764.194,A -85,B 0,C 180,E1 -14828.512,E2 -14828.512} C_VEL
LIN {X 0,Y 334.608,Z 776.291,A -85,B 0,C 180,E1 -14829.242,E2 -14829.242} C_VEL
LIN {X 0,Y 333.154,Z 788.861,A -85,B 0,C 180,E1 -14830.274,E2 -14830.274} C_VEL
LIN {X 0,Y 331.657,Z 800.143,A -85,B 0,C 180,E1 -14831.467,E2 -14831.467} C_VEL
LIN {X 0,Y 330.169,Z 810.469,A -85,B 0,C 180,E1 -14832.838,E2 -14832.838} C_VEL
LIN {X 0,Y 328.717,Z 820.821,A -85,B 0,C 180,E1 -14834.572,E2 -14834.572} C_VEL
LIN {X 0,Y 327.483,Z 829.373,A -85,B 0,C 180,E1 -14836.346,E2 -14836.346} C_VEL
LIN {X 0,Y 326.366,Z 836.534,A -85,B 0,C 180,E1 -14838.196,E2 -14838.196} C_VEL
LIN {X 0,Y 325.699,Z 842.292,A -85,B 0,C 180,E1 -14840.06,E2 -14840.06} C_VEL
LIN {X 0,Y 325.237,Z 846.839,A -85,B 0,C 180,E1 -14841.926,E2 -14841.926} C_VEL
LIN {X 0,Y 325.02,Z 850.741,A -85,B 0,C 180,E1 -14844.087,E2 -14844.087} C_VEL
LIN {X 0,Y 324.958,Z 853.356,A -85,B 0,C 180,E1 -14846.28,E2 -14846.28} C_VEL
LIN {X 0,Y 324.916,Z 854.251,A -85,B 0,C 180,E1 -14847.521,E2 -14847.521} C_VEL
LIN {X 0,Y 324.974,Z 854.71,A -85,B 0,C 180,E1 -14848.761,E2 -14848.761} C_VEL
LIN {X 0,Y 325.071,Z 854.771,A -85,B 0,C 180,E1 -14850,E2 -14850} C_VEL
LIN {X 0,Y 325.006,Z 854.425,A -85,B 0,C 180,E1 -14851.239,E2 -14851.239} C_VEL
LIN {X 0,Y 324.927,Z 853.647,A -85,B 0,C 180,E1 -14852.479,E2 -14852.479} C_VEL
LIN {X 0,Y 324.96,Z 852.426,A -85,B 0,C 180,E1 -14853.72,E2 -14853.72} C_VEL
LIN {X 0,Y 325.024,Z 849.208,A -85,B 0,C 180,E1 -14855.919,E2 -14855.919} C_VEL
LIN {X 0,Y 325.236,Z 844.638,A -85,B 0,C 180,E1 -14858.074,E2 -14858.074} C_VEL
LIN {X 0,Y 325.717,Z 838.343,A -85,B 0,C 180,E1 -14860.254,E2 -14860.254} C_VEL
LIN {X 0,Y 326.429,Z 831.468,A -85,B 0,C 180,E1 -14862.117,E2 -14862.117} C_VEL
LIN {X 0,Y 327.242,Z 824.446,A -85,B 0,C 180,E1 -14863.664,E2 -14863.664} C_VEL
LIN {X 0,Y 328.202,Z 816.357,A -85,B 0,C 180,E1 -14865.141,E2 -14865.141} C_VEL
LIN {X 0,Y 329.205,Z 806.705,A -85,B 0,C 180,E1 -14866.59,E2 -14866.59} C_VEL
LIN {X 0,Y 330.352,Z 796.634,A -85,B 0,C 180,E1 -14867.807,E2 -14867.807} C_VEL
LIN {X 0,Y 331.523,Z 785.717,A -85,B 0,C 180,E1 -14868.861,E2 -14868.861} C_VEL
LIN {X 0,Y 332.582,Z 773.722,A -85,B 0,C 180,E1 -14869.761,E2 -14869.761} C_VEL
LIN {X 0,Y 333.554,Z 760.745,A -85,B 0,C 180,E1 -14870.464,E2 -14870.464} C_VEL
LIN {X 0,Y 334.146,Z 746.739,A -85,B 0,C 180,E1 -14870.95,E2 -14870.95} C_VEL
LIN {X 0,Y 335.62,Z 682.009,A -85,B 0,C 180,E1 -14872.453,E2 -14872.453} C_VEL
LIN {X 0,Y 330.009,Z 642.443,A -85,B 0,C 180,E1 -14873.818,E2 -14873.818} C_VEL
LIN {X 0,Y 331.196,Z 632.975,A -85,B 0,C 180,E1 -14876.123,E2 -14876.123} C_VEL
LIN {X 0,Y 330.182,Z 626.164,A -85,B 0,C 180,E1 -14877.922,E2 -14877.922} C_VEL
LIN {X 0,Y 327.171,Z 612.397,A -85,B 0,C 180,E1 -14881.754,E2 -14881.754} C_VEL
LIN {X 0,Y 326.609,Z 609.804,A -85,B 0,C 180,E1 -14882.543,E2 -14882.543} C_VEL
LIN {X 0,Y 326.612,Z 609.797,A -85,B 0,C 180,E1 -14885.519,E2 -14885.519} C_VEL
LIN {X 0,Y 326.634,Z 609.795,A -85,B 0,C 180,E1 -14889.231,E2 -14889.231} C_VEL
LIN {X 0,Y 326.612,Z 609.8,A -85,B 0,C 180,E1 -14892.978,E2 -14892.978} C_VEL
LIN {X 0,Y 326.603,Z 609.801,A -85,B 0,C 180,E1 -14897.022,E2 -14897.022} C_VEL
LIN {X 0,Y 326.632,Z 609.801,A -85,B 0,C 180,E1 -14900.767,E2 -14900.767} C_VEL
LIN {X 0,Y 326.61,Z 609.8,A -85,B 0,C 180,E1 -14904.479,E2 -14904.479} C_VEL
LIN {X 0,Y 326.611,Z 609.798,A -85,B 0,C 180,E1 -14907.455,E2 -14907.455} C_VEL
LIN {X 0,Y 326.657,Z 609.793,A -85,B 0,C 180,E1 -14910.34,E2 -14910.34} C_VEL
LIN {X 0,Y 326.685,Z 609.79,A -85,B 0,C 180,E1 -14914.515,E2 -14914.515} C_VEL
LIN {X 0,Y 326.614,Z 609.798,A -85,B 0,C 180,E1 -14918.542,E2 -14918.542} C_VEL
LIN {X 0,Y 326.739,Z 609.787,A -85,B 0,C 180,E1 -14921.177,E2 -14921.177} C_VEL
LIN {X 0,Y 326.757,Z 609.783,A -85,B 0,C 180,E1 -14925.432,E2 -14925.432} C_VEL
LIN {X 0,Y 326.763,Z 609.781,A -85,B 0,C 180,E1 -14928.838,E2 -14928.838} C_VEL
LIN {X 0,Y 326.96,Z 609.754,A -85,B 0,C 180,E1 -14932.589,E2 -14932.589} C_VEL
LIN {X 0,Y 326.772,Z 609.78,A -85,B 0,C 180,E1 -14935.064,E2 -14935.064} C_VEL
LIN {X 0,Y 327.04,Z 609.749,A -85,B 0,C 180,E1 -14937.536,E2 -14937.536} C_VEL
LIN {X 0,Y 327.21,Z 609.724,A -85,B 0,C 180,E1 -14939.999,E2 -14939.999} C_VEL
LIN {X 0,Y 327.041,Z 609.743,A -85,B 0,C 180,E1 -14942.463,E2 -14942.463} C_VEL
LIN {X 0,Y 326.959,Z 609.754,A -85,B 0,C 180,E1 -14946.625,E2 -14946.625} C_VEL
LIN {X 0,Y 326.805,Z 609.776,A -85,B 0,C 180,E1 -14949.906,E2 -14949.906} C_VEL
LIN {X 0,Y 326.751,Z 609.785,A -85,B 0,C 180,E1 -14953.685,E2 -14953.685} C_VEL
LIN {X 0,Y 326.69,Z 609.791,A -85,B 0,C 180,E1 -14957.528,E2 -14957.528} C_VEL
LIN {X 0,Y 326.654,Z 609.795,A -85,B 0,C 180,E1 -14960.135,E2 -14960.135} C_VEL
LIN {X 0,Y 326.643,Z 609.796,A -85,B 0,C 180,E1 -14964.129,E2 -14964.129} C_VEL
LIN {X 0,Y 326.677,Z 609.789,A -85,B 0,C 180,E1 -14966.858,E2 -14966.858} C_VEL
LIN {X 0,Y 326.634,Z 609.795,A -85,B 0,C 180,E1 -14970.612,E2 -14970.612} C_VEL
LIN {X 0,Y 326.601,Z 609.804,A -85,B 0,C 180,E1 -14974.019,E2 -14974.019} C_VEL
LIN {X 0,Y 326.622,Z 609.795,A -85,B 0,C 180,E1 -14977.239,E2 -14977.239} C_VEL
LIN {X 0,Y 326.628,Z 609.801,A -85,B 0,C 180,E1 -14980.203,E2 -14980.203} C_VEL
LIN {X 0,Y 326.623,Z 609.796,A -85,B 0,C 180,E1 -14983.514,E2 -14983.514} C_VEL
LIN {X 0,Y 326.61,Z 609.798,A -85,B 0,C 180,E1 -14987.021,E2 -14987.021} C_VEL
LIN {X 0,Y 326.635,Z 609.794,A -85,B 0,C 180,E1 -14991.394,E2 -14991.394} C_VEL
LIN {X 0,Y 326.614,Z 609.799,A -85,B 0,C 180,E1 -14994.851,E2 -14994.851} C_VEL
LIN {X 0,Y 326.602,Z 609.798,A -85,B 0,C 180,E1 -14997.456,E2 -14997.456} C_VEL
LIN {X 0,Y 326.642,Z 609.797,A -85,B 0,C 180,E1 -15000.34,E2 -15000.34} C_VEL
LIN {X 0,Y 326.685,Z 609.793,A -85,B 0,C 180,E1 -15004.517,E2 -15004.517} C_VEL
LIN {X 0,Y 326.644,Z 609.798,A -85,B 0,C 180,E1 -15008.546,E2 -15008.546} C_VEL
LIN {X 0,Y 326.74,Z 609.783,A -85,B 0,C 180,E1 -15011.178,E2 -15011.178} C_VEL
LIN {X 0,Y 326.759,Z 609.78,A -85,B 0,C 180,E1 -15015.433,E2 -15015.433} C_VEL
LIN {X 0,Y 326.766,Z 609.784,A -85,B 0,C 180,E1 -15018.839,E2 -15018.839} C_VEL
LIN {X 0,Y 326.963,Z 609.756,A -85,B 0,C 180,E1 -15022.59,E2 -15022.59} C_VEL
LIN {X 0,Y 326.774,Z 609.782,A -85,B 0,C 180,E1 -15025.065,E2 -15025.065} C_VEL
LIN {X 0,Y 327.045,Z 609.745,A -85,B 0,C 180,E1 -15027.537,E2 -15027.537} C_VEL
LIN {X 0,Y 327.196,Z 609.724,A -85,B 0,C 180,E1 -15030,E2 -15030} C_VEL
LIN {X 0,Y 327.045,Z 609.744,A -85,B 0,C 180,E1 -15032.463,E2 -15032.463} C_VEL
LIN {X 0,Y 326.986,Z 609.751,A -85,B 0,C 180,E1 -15036.169,E2 -15036.169} C_VEL
LIN {X 0,Y 326.802,Z 609.774,A -85,B 0,C 180,E1 -15039.906,E2 -15039.906} C_VEL
LIN {X 0,Y 326.755,Z 609.782,A -85,B 0,C 180,E1 -15043.685,E2 -15043.685} C_VEL
LIN {X 0,Y 326.7,Z 609.792,A -85,B 0,C 180,E1 -15047.527,E2 -15047.527} C_VEL
LIN {X 0,Y 326.677,Z 609.802,A -85,B 0,C 180,E1 -15050.134,E2 -15050.134} C_VEL
LIN {X 0,Y 327.265,Z 612.816,A -85,B 0,C 180,E1 -15051.123,E2 -15051.123} C_VEL
LIN {X 0,Y 335.462,Z 635.88,A -85,B 0,C 180,E1 -15052.243,E2 -15052.243} C_VEL
LIN {X 0,Y 336.313,Z 641.246,A -85,B 0,C 180,E1 -15052.428,E2 -15052.428} C_VEL
LIN {X 0,Y 334.258,Z 720.518,A -85,B 0,C 180,E1 -15054.287,E2 -15054.287} C_VEL
LIN {X 0,Y 333.646,Z 734.321,A -85,B 0,C 180,E1 -15054.873,E2 -15054.873} C_VEL
LIN {X 0,Y 332.84,Z 747.057,A -85,B 0,C 180,E1 -15055.674,E2 -15055.674} C_VEL
LIN {X 0,Y 331.929,Z 757.747,A -85,B 0,C 180,E1 -15056.561,E2 -15056.561} C_VEL
LIN {X 0,Y 330.89,Z 769.031,A -85,B 0,C 180,E1 -15057.754,E2 -15057.754} C_VEL
LIN {X 0,Y 329.731,Z 779.191,A -85,B 0,C 180,E1 -15059.088,E2 -15059.088} C_VEL
LIN {X 0,Y 328.644,Z 788.998,A -85,B 0,C 180,E1 -15060.7,E2 -15060.7} C_VEL
LIN {X 0,Y 327.605,Z 797.512,A -85,B 0,C 180,E1 -15062.432,E2 -15062.432} C_VEL
LIN {X 0,Y 326.86,Z 803.768,A -85,B 0,C 180,E1 -15063.989,E2 -15063.989} C_VEL
LIN {X 0,Y 326.135,Z 810.117,A -85,B 0,C 180,E1 -15065.937,E2 -15065.937} C_VEL
LIN {X 0,Y 325.595,Z 815.226,A -85,B 0,C 180,E1 -15067.963,E2 -15067.963} C_VEL
LIN {X 0,Y 325.224,Z 818.455,A -85,B 0,C 180,E1 -15069.649,E2 -15069.649} C_VEL
LIN {X 0,Y 325.035,Z 820.203,A -85,B 0,C 180,E1 -15070.82,E2 -15070.82} C_VEL
LIN {X 0,Y 324.86,Z 822.164,A -85,B 0,C 180,E1 -15072.647,E2 -15072.647} C_VEL
LIN {X 0,Y 324.75,Z 823.194,A -85,B 0,C 180,E1 -15074.427,E2 -15074.427} C_VEL
LIN {X 0,Y 324.779,Z 823.395,A -85,B 0,C 180,E1 -15076.176,E2 -15076.176} C_VEL
LIN {X 0,Y 324.932,Z 822.826,A -85,B 0,C 180,E1 -15077.891,E2 -15077.891} C_VEL
LIN {X 0,Y 324.416,Z 822.197,A -85,B 0,C 180,E1 -15078.922,E2 -15078.922} C_VEL
LIN {X 0,Y 321.853,Z 820.657,A -85,B 0,C 180,E1 -15080.598,E2 -15080.598} C_VEL
LIN {X 0,Y 319.751,Z 818.945,A -85,B 0,C 180,E1 -15081.937,E2 -15081.937} C_VEL
LIN {X 0,Y 319.015,Z 817.306,A -85,B 0,C 180,E1 -15082.952,E2 -15082.952} C_VEL
LIN {X 0,Y 319.047,Z 816.655,A -85,B 0,C 180,E1 -15083.29,E2 -15083.29} C_VEL
LIN {X 0,Y 319.772,Z 812.468,A -85,B 0,C 180,E1 -15085.151,E2 -15085.151} C_VEL
LIN {X 0,Y 320.739,Z 806.646,A -85,B 0,C 180,E1 -15087.159,E2 -15087.159} C_VEL
LIN {X 0,Y 322.069,Z 799.01,A -85,B 0,C 180,E1 -15089.202,E2 -15089.202} C_VEL
LIN {X 0,Y 323.559,Z 790.596,A -85,B 0,C 180,E1 -15090.984,E2 -15090.984} C_VEL
LIN {X 0,Y 324.876,Z 781.889,A -85,B 0,C 180,E1 -15092.489,E2 -15092.489} C_VEL
LIN {X 0,Y 326.233,Z 772.634,A -85,B 0,C 180,E1 -15093.794,E2 -15093.794} C_VEL
LIN {X 0,Y 327.54,Z 762.734,A -85,B 0,C 180,E1 -15094.928,E2 -15094.928} C_VEL
LIN {X 0,Y 328.902,Z 750.296,A -85,B 0,C 180,E1 -15096.047,E2 -15096.047} C_VEL
LIN {X 0,Y 329.96,Z 737.779,A -85,B 0,C 180,E1 -15096.896,E2 -15096.896} C_VEL
LIN {X 0,Y 330.632,Z 726.297,A -85,B 0,C 180,E1 -15097.453,E2 -15097.453} C_VEL
LIN {X 0,Y 331.267,Z 710.559,A -85,B 0,C 180,E1 -15097.912,E2 -15097.912} C_VEL
LIN {X 0,Y 333.346,Z 643.548,A -85,B 0,C 180,E1 -15099.549,E2 -15099.549} C_VEL
LIN {X 0,Y 326.861,Z 628.23,A -85,B 0,C 180,E1 -15100.638,E2 -15100.638} C_VEL
LIN {X 0,Y 320.871,Z 615.701,A -85,B 0,C 180,E1 -15101.69,E2 -15101.69} C_VEL
LIN {X 0,Y 319.696,Z 610.662,A -85,B 0,C 180,E1 -15103.805,E2 -15103.805} C_VEL
LIN {X 0,Y 319.677,Z 610.665,A -85,B 0,C 180,E1 -15107.301,E2 -15107.301} C_VEL
LIN {X 0,Y 319.874,Z 610.643,A -85,B 0,C 180,E1 -15111.37,E2 -15111.37} C_VEL
LIN {X 0,Y 319.947,Z 610.632,A -85,B 0,C 180,E1 -15113.695,E2 -15113.695} C_VEL
LIN {X 0,Y 320.011,Z 610.624,A -85,B 0,C 180,E1 -15117.483,E2 -15117.483} C_VEL
LIN {X 0,Y 320.162,Z 610.604,A -85,B 0,C 180,E1 -15120.001,E2 -15120.001} C_VEL
LIN {X 0,Y 320.002,Z 610.625,A -85,B 0,C 180,E1 -15122.518,E2 -15122.518} C_VEL
LIN {X 0,Y 319.948,Z 610.629,A -85,B 0,C 180,E1 -15126.306,E2 -15126.306} C_VEL
LIN {X 0,Y 319.836,Z 610.644,A -85,B 0,C 180,E1 -15128.849,E2 -15128.849} C_VEL
LIN {X 0,Y 319.678,Z 610.66,A -85,B 0,C 180,E1 -15132.701,E2 -15132.701} C_VEL
LIN {X 0,Y 319.693,Z 610.658,A -85,B 0,C 180,E1 -15135.296,E2 -15135.296} C_VEL
LIN {X 0,Y 319.669,Z 610.661,A -85,B 0,C 180,E1 -15139.256,E2 -15139.256} C_VEL
LIN {X 0,Y 319.565,Z 610.675,A -85,B 0,C 180,E1 -15143.32,E2 -15143.32} C_VEL
LIN {X 0,Y 319.63,Z 610.663,A -85,B 0,C 180,E1 -15146.089,E2 -15146.089} C_VEL
LIN {X 0,Y 319.585,Z 610.668,A -85,B 0,C 180,E1 -15148.935,E2 -15148.935} C_VEL
LIN {X 0,Y 319.535,Z 610.673,A -85,B 0,C 180,E1 -15151.862,E2 -15151.862} C_VEL
LIN {X 0,Y 319.576,Z 610.671,A -85,B 0,C 180,E1 -15155.544,E2 -15155.544} C_VEL
LIN {X 0,Y 319.578,Z 610.67,A -85,B 0,C 180,E1 -15158.008,E2 -15158.008} C_VEL
LIN {X 0,Y 319.566,Z 610.677,A -85,B 0,C 180,E1 -15161.607,E2 -15161.607} C_VEL
LIN {X 0,Y 319.553,Z 610.68,A -85,B 0,C 180,E1 -15165.27,E2 -15165.27} C_VEL
LIN {X 0,Y 319.545,Z 610.682,A -85,B 0,C 180,E1 -15168.716,E2 -15168.716} C_VEL
LIN {X 0,Y 319.582,Z 610.678,A -85,B 0,C 180,E1 -15172.344,E2 -15172.344} C_VEL
LIN {X 0,Y 319.593,Z 610.726,A -85,B 0,C 180,E1 -15174.543,E2 -15174.543} C_VEL
LIN {X 0,Y 321.899,Z 619.732,A -85,B 0,C 180,E1 -15177.664,E2 -15177.664} C_VEL
LIN {X 0,Y 324.127,Z 629.75,A -85,B 0,C 180,E1 -15180.867,E2 -15180.867} C_VEL
LIN {X 0,Y 325.419,Z 637,A -85,B 0,C 180,E1 -15183.03,E2 -15183.03} C_VEL
LIN {X 0,Y 325.047,Z 639.909,A -85,B 0,C 180,E1 -15183.795,E2 -15183.795} C_VEL
LIN {X 0,Y 329.679,Z 663.634,A -85,B 0,C 180,E1 -15184.958,E2 -15184.958} C_VEL
LIN {X 0,Y 332.336,Z 683.221,A -85,B 0,C 180,E1 -15185.749,E2 -15185.749} C_VEL
LIN {X 0,Y 330.526,Z 744.706,A -85,B 0,C 180,E1 -15187.254,E2 -15187.254} C_VEL
LIN {X 0,Y 329.771,Z 758.385,A -85,B 0,C 180,E1 -15187.732,E2 -15187.732} C_VEL
LIN {X 0,Y 328.601,Z 771.424,A -85,B 0,C 180,E1 -15188.433,E2 -15188.433} C_VEL
LIN {X 0,Y 327.124,Z 784.313,A -85,B 0,C 180,E1 -15189.403,E2 -15189.403} C_VEL
LIN {X 0,Y 325.722,Z 795.116,A -85,B 0,C 180,E1 -15190.462,E2 -15190.462} C_VEL
LIN {X 0,Y 324.067,Z 806.222,A -85,B 0,C 180,E1 -15191.836,E2 -15191.836} C_VEL
LIN {X 0,Y 322.687,Z 815.276,A -85,B 0,C 180,E1 -15193.227,E2 -15193.227} C_VEL
LIN {X 0,Y 321.179,Z 825.139,A -85,B 0,C 180,E1 -15195.102,E2 -15195.102} C_VEL
LIN {X 0,Y 319.961,Z 833.046,A -85,B 0,C 180,E1 -15196.989,E2 -15196.989} C_VEL
LIN {X 0,Y 319.084,Z 838.467,A -85,B 0,C 180,E1 -15198.567,E2 -15198.567} C_VEL
LIN {X 0,Y 318.476,Z 843.756,A -85,B 0,C 180,E1 -15200.474,E2 -15200.474} C_VEL
LIN {X 0,Y 318.066,Z 847.893,A -85,B 0,C 180,E1 -15202.382,E2 -15202.382} C_VEL
LIN {X 0,Y 317.91,Z 850.796,A -85,B 0,C 180,E1 -15204.165,E2 -15204.165} C_VEL
LIN {X 0,Y 317.862,Z 853.066,A -85,B 0,C 180,E1 -15206.197,E2 -15206.197} C_VEL
LIN {X 0,Y 317.834,Z 853.927,A -85,B 0,C 180,E1 -15207.465,E2 -15207.465} C_VEL
LIN {X 0,Y 317.878,Z 854.368,A -85,B 0,C 180,E1 -15208.733,E2 -15208.733} C_VEL
LIN {X 0,Y 317.979,Z 854.413,A -85,B 0,C 180,E1 -15210,E2 -15210} C_VEL
LIN {X 0,Y 317.91,Z 854.049,A -85,B 0,C 180,E1 -15211.267,E2 -15211.267} C_VEL
LIN {X 0,Y 317.844,Z 853.234,A -85,B 0,C 180,E1 -15212.535,E2 -15212.535} C_VEL
LIN {X 0,Y 317.887,Z 851.994,A -85,B 0,C 180,E1 -15213.803,E2 -15213.803} C_VEL
LIN {X 0,Y 317.921,Z 849.068,A -85,B 0,C 180,E1 -15215.854,E2 -15215.854} C_VEL
LIN {X 0,Y 318.067,Z 845.574,A -85,B 0,C 180,E1 -15217.618,E2 -15217.618} C_VEL
LIN {X 0,Y 318.44,Z 840.675,A -85,B 0,C 180,E1 -15219.528,E2 -15219.528} C_VEL
LIN {X 0,Y 318.985,Z 834.463,A -85,B 0,C 180,E1 -15221.437,E2 -15221.437} C_VEL
LIN {X 0,Y 319.989,Z 826.737,A -85,B 0,C 180,E1 -15223.333,E2 -15223.333} C_VEL
LIN {X 0,Y 320.938,Z 818.796,A -85,B 0,C 180,E1 -15224.91,E2 -15224.91} C_VEL
LIN {X 0,Y 321.93,Z 809.067,A -85,B 0,C 180,E1 -15226.487,E2 -15226.487} C_VEL
LIN {X 0,Y 323.269,Z 798.319,A -85,B 0,C 180,E1 -15227.883,E2 -15227.883} C_VEL
LIN {X 0,Y 324.427,Z 787.948,A -85,B 0,C 180,E1 -15228.962,E2 -15228.962} C_VEL
LIN {X 0,Y 325.597,Z 775.583,A -85,B 0,C 180,E1 -15229.956,E2 -15229.956} C_VEL
LIN {X 0,Y 326.612,Z 762.723,A -85,B 0,C 180,E1 -15230.713,E2 -15230.713} C_VEL
LIN {X 0,Y 327.274,Z 750.48,A -85,B 0,C 180,E1 -15231.205,E2 -15231.205} C_VEL
LIN {X 0,Y 328.897,Z 682.883,A -85,B 0,C 180,E1 -15232.827,E2 -15232.827} C_VEL
LIN {X 0,Y 323.191,Z 642.201,A -85,B 0,C 180,E1 -15234.249,E2 -15234.249} C_VEL
LIN {X 0,Y 324.243,Z 633.66,A -85,B 0,C 180,E1 -15236.38,E2 -15236.38} C_VEL
LIN {X 0,Y 322.737,Z 625.463,A -85,B 0,C 180,E1 -15238.624,E2 -15238.624} C_VEL
LIN {X 0,Y 320.072,Z 613.045,A -85,B 0,C 180,E1 -15242.172,E2 -15242.172} C_VEL
LIN {X 0,Y 319.57,Z 610.68,A -85,B 0,C 180,E1 -15242.882,E2 -15242.882} C_VEL
LIN {X 0,Y 319.559,Z 610.681,A -85,B 0,C 180,E1 -15246.426,E2 -15246.426} C_VEL
LIN {X 0,Y 319.563,Z 610.676,A -85,B 0,C 180,E1 -15249.669,E2 -15249.669} C_VEL
LIN {X 0,Y 319.581,Z 610.674,A -85,B 0,C 180,E1 -15253.471,E2 -15253.471} C_VEL
LIN {X 0,Y 319.579,Z 610.676,A -85,B 0,C 180,E1 -15257.02,E2 -15257.02} C_VEL
LIN {X 0,Y 319.579,Z 610.676,A -85,B 0,C 180,E1 -15260.375,E2 -15260.375} C_VEL
LIN {X 0,Y 319.558,Z 610.677,A -85,B 0,C 180,E1 -15263.572,E2 -15263.572} C_VEL
LIN {X 0,Y 319.575,Z 610.678,A -85,B 0,C 180,E1 -15266.685,E2 -15266.685} C_VEL
LIN {X 0,Y 319.589,Z 610.672,A -85,B 0,C 180,E1 -15269.616,E2 -15269.616} C_VEL
LIN {X 0,Y 319.604,Z 610.672,A -85,B 0,C 180,E1 -15272.497,E2 -15272.497} C_VEL
LIN {X 0,Y 319.598,Z 610.674,A -85,B 0,C 180,E1 -15275.303,E2 -15275.303} C_VEL
LIN {X 0,Y 319.596,Z 610.674,A -85,B 0,C 180,E1 -15279.399,E2 -15279.399} C_VEL
LIN {X 0,Y 319.652,Z 610.664,A -85,B 0,C 180,E1 -15282.072,E2 -15282.072} C_VEL
LIN {X 0,Y 319.726,Z 610.656,A -85,B 0,C 180,E1 -15286.007,E2 -15286.007} C_VEL
LIN {X 0,Y 319.75,Z 610.652,A -85,B 0,C 180,E1 -15289.872,E2 -15289.872} C_VEL
LIN {X 0,Y 319.919,Z 610.631,A -85,B 0,C 180,E1 -15292.425,E2 -15292.425} C_VEL
LIN {X 0,Y 319.741,Z 610.655,A -85,B 0,C 180,E1 -15294.955,E2 -15294.955} C_VEL
LIN {X 0,Y 319.984,Z 610.628,A -85,B 0,C 180,E1 -15297.482,E2 -15297.482} C_VEL
LIN {X 0,Y 320.161,Z 610.601,A -85,B 0,C 180,E1 -15299.999,E2 -15299.999} C_VEL
LIN {X 0,Y 319.985,Z 610.622,A -85,B 0,C 180,E1 -15302.517,E2 -15302.517} C_VEL
LIN {X 0,Y 319.921,Z 610.631,A -85,B 0,C 180,E1 -15306.614,E2 -15306.614} C_VEL
LIN {X 0,Y 319.835,Z 610.642,A -85,B 0,C 180,E1 -15308.848,E2 -15308.848} C_VEL
LIN {X 0,Y 319.673,Z 610.66,A -85,B 0,C 180,E1 -15312.7,E2 -15312.7} C_VEL
LIN {X 0,Y 319.691,Z 610.66,A -85,B 0,C 180,E1 -15315.295,E2 -15315.295} C_VEL
LIN {X 0,Y 319.666,Z 610.664,A -85,B 0,C 180,E1 -15319.255,E2 -15319.255} C_VEL
LIN {X 0,Y 319.562,Z 610.676,A -85,B 0,C 180,E1 -15323.319,E2 -15323.319} C_VEL
LIN {X 0,Y 319.627,Z 610.671,A -85,B 0,C 180,E1 -15326.088,E2 -15326.088} C_VEL
LIN {X 0,Y 319.582,Z 610.673,A -85,B 0,C 180,E1 -15328.934,E2 -15328.934} C_VEL
LIN {X 0,Y 319.531,Z 610.684,A -85,B 0,C 180,E1 -15331.861,E2 -15331.861} C_VEL
LIN {X 0,Y 319.572,Z 610.675,A -85,B 0,C 180,E1 -15335.543,E2 -15335.543} C_VEL
LIN {X 0,Y 319.592,Z 610.675,A -85,B 0,C 180,E1 -15338.004,E2 -15338.004} C_VEL
LIN {X 0,Y 319.59,Z 610.673,A -85,B 0,C 180,E1 -15341.612,E2 -15341.612} C_VEL
LIN {X 0,Y 319.575,Z 610.674,A -85,B 0,C 180,E1 -15345.274,E2 -15345.274} C_VEL
LIN {X 0,Y 319.54,Z 610.679,A -85,B 0,C 180,E1 -15348.715,E2 -15348.715} C_VEL
LIN {X 0,Y 319.576,Z 610.679,A -85,B 0,C 180,E1 -15352.343,E2 -15352.343} C_VEL
LIN {X 0,Y 319.554,Z 610.677,A -85,B 0,C 180,E1 -15355.124,E2 -15355.124} C_VEL
LIN {X 0,Y 319.561,Z 610.676,A -85,B 0,C 180,E1 -15359.06,E2 -15359.06} C_VEL
LIN {X 0,Y 319.601,Z 610.676,A -85,B 0,C 180,E1 -15362.498,E2 -15362.498} C_VEL
LIN {X 0,Y 319.6,Z 610.671,A -85,B 0,C 180,E1 -15365.304,E2 -15365.304} C_VEL
LIN {X 0,Y 319.593,Z 610.672,A -85,B 0,C 180,E1 -15368.048,E2 -15368.048} C_VEL
LIN {X 0,Y 319.685,Z 610.664,A -85,B 0,C 180,E1 -15370.963,E2 -15370.963} C_VEL
LIN {X 0,Y 319.727,Z 610.656,A -85,B 0,C 180,E1 -15375.276,E2 -15375.276} C_VEL
LIN {X 0,Y 319.754,Z 610.651,A -85,B 0,C 180,E1 -15379.873,E2 -15379.873} C_VEL
LIN {X 0,Y 319.922,Z 610.632,A -85,B 0,C 180,E1 -15382.426,E2 -15382.426} C_VEL
LIN {X 0,Y 319.743,Z 610.659,A -85,B 0,C 180,E1 -15384.956,E2 -15384.956} C_VEL
LIN {X 0,Y 319.989,Z 610.624,A -85,B 0,C 180,E1 -15387.482,E2 -15387.482} C_VEL
LIN {X 0,Y 320.148,Z 610.602,A -85,B 0,C 180,E1 -15390,E2 -15390} C_VEL
LIN {X 0,Y 319.989,Z 610.623,A -85,B 0,C 180,E1 -15392.518,E2 -15392.518} C_VEL
LIN {X 0,Y 319.94,Z 610.628,A -85,B 0,C 180,E1 -15396.306,E2 -15396.306} C_VEL
LIN {X 0,Y 319.834,Z 610.644,A -85,B 0,C 180,E1 -15398.848,E2 -15398.848} C_VEL
LIN {X 0,Y 319.678,Z 610.662,A -85,B 0,C 180,E1 -15402.7,E2 -15402.7} C_VEL
LIN {X 0,Y 319.696,Z 610.665,A -85,B 0,C 180,E1 -15405.295,E2 -15405.295} C_VEL
LIN {X 0,Y 319.678,Z 610.667,A -85,B 0,C 180,E1 -15409.588,E2 -15409.588} C_VEL
LIN {X 0,Y 319.699,Z 610.968,A -85,B 0,C 180,E1 -15409.921,E2 -15409.921} C_VEL
LIN {X 0,Y 320.112,Z 613.139,A -85,B 0,C 180,E1 -15410.649,E2 -15410.649} C_VEL
LIN {X 0,Y 329.082,Z 638.379,A -85,B 0,C 180,E1 -15411.904,E2 -15411.904} C_VEL
LIN {X 0,Y 329.608,Z 642.119,A -85,B 0,C 180,E1 -15412.032,E2 -15412.032} C_VEL
LIN {X 0,Y 327.489,Z 720.787,A -85,B 0,C 180,E1 -15413.918,E2 -15413.918} C_VEL
LIN {X 0,Y 326.869,Z 734.884,A -85,B 0,C 180,E1 -15414.533,E2 -15414.533} C_VEL
LIN {X 0,Y 326.036,Z 747.188,A -85,B 0,C 180,E1 -15415.32,E2 -15415.32} C_VEL
LIN {X 0,Y 325.053,Z 758.767,A -85,B 0,C 180,E1 -15416.31,E2 -15416.31} C_VEL
LIN {X 0,Y 323.95,Z 769.73,A -85,B 0,C 180,E1 -15417.5,E2 -15417.5} C_VEL
LIN {X 0,Y 322.709,Z 780.498,A -85,B 0,C 180,E1 -15418.968,E2 -15418.968} C_VEL
LIN {X 0,Y 321.53,Z 790.701,A -85,B 0,C 180,E1 -15420.725,E2 -15420.725} C_VEL
LIN {X 0,Y 320.453,Z 799.021,A -85,B 0,C 180,E1 -15422.5,E2 -15422.5} C_VEL
LIN {X 0,Y 319.57,Z 806.44,A -85,B 0,C 180,E1 -15424.5,E2 -15424.5} C_VEL
LIN {X 0,Y 318.905,Z 812.329,A -85,B 0,C 180,E1 -15426.513,E2 -15426.513} C_VEL
LIN {X 0,Y 318.324,Z 817.343,A -85,B 0,C 180,E1 -15428.766,E2 -15428.766} C_VEL
LIN {X 0,Y 318.109,Z 819.18,A -85,B 0,C 180,E1 -15429.843,E2 -15429.843} C_VEL
LIN {X 0,Y 317.874,Z 821.442,A -85,B 0,C 180,E1 -15431.549,E2 -15431.549} C_VEL
LIN {X 0,Y 317.732,Z 822.941,A -85,B 0,C 180,E1 -15433.289,E2 -15433.289} C_VEL
LIN {X 0,Y 317.647,Z 823.694,A -85,B 0,C 180,E1 -15435.072,E2 -15435.072} C_VEL
LIN {X 0,Y 317.751,Z 823.652,A -85,B 0,C 180,E1 -15436.876,E2 -15436.876} C_VEL
LIN {X 0,Y 317.951,Z 822.757,A -85,B 0,C 180,E1 -15438.722,E2 -15438.722} C_VEL
LIN {X 0,Y 318.343,Z 820.937,A -85,B 0,C 180,E1 -15440.594,E2 -15440.594} C_VEL
LIN {X 0,Y 318.809,Z 818.1,A -85,B 0,C 180,E1 -15442.522,E2 -15442.522} C_VEL
LIN {X 0,Y 319.047,Z 816.655,A -85,B 0,C 180,E1 -15443.29,E2 -15443.29} C_VEL
LIN {X 0,Y 318.757,Z 814.699,A -85,B 0,C 180,E1 -15444.29,E2 -15444.29} C_VEL
LIN {X 0,Y 316.61,Z 811.125,A -85,B 0,C 180,E1 -15445.914,E2 -15445.914} C_VEL
LIN {X 0,Y 314.581,Z 806.886,A -85,B 0,C 180,E1 -15447.501,E2 -15447.501} C_VEL
LIN {X 0,Y 314.477,Z 803.853,A -85,B 0,C 180,E1 -15448.428,E2 -15448.428} C_VEL
LIN {X 0,Y 315.787,Z 796.697,A -85,B 0,C 180,E1 -15450.22,E2 -15450.22} C_VEL
LIN {X 0,Y 317.299,Z 788.252,A -85,B 0,C 180,E1 -15451.923,E2 -15451.923} C_VEL
LIN {X 0,Y 318.8,Z 778.734,A -85,B 0,C 180,E1 -15453.487,E2 -15453.487} C_VEL
LIN {X 0,Y 320.332,Z 768.23,A -85,B 0,C 180,E1 -15454.874,E2 -15454.874} C_VEL
LIN {X 0,Y 321.815,Z 757.114,A -85,B 0,C 180,E1 -15456.024,E2 -15456.024} C_VEL
LIN {X 0,Y 323.102,Z 744.487,A -85,B 0,C 180,E1 -15457.036,E2 -15457.036} C_VEL
LIN {X 0,Y 323.964,Z 731.616,A -85,B 0,C 180,E1 -15457.794,E2 -15457.794} C_VEL
LIN {X 0,Y 324.692,Z 718.386,A -85,B 0,C 180,E1 -15458.285,E2 -15458.285} C_VEL
LIN {X 0,Y 327.142,Z 645.434,A -85,B 0,C 180,E1 -15460.11,E2 -15460.11} C_VEL
LIN {X 0,Y 320.249,Z 629.347,A -85,B 0,C 180,E1 -15461.322,E2 -15461.322} C_VEL
LIN {X 0,Y 313.748,Z 616.259,A -85,B 0,C 180,E1 -15462.483,E2 -15462.483} C_VEL
LIN {X 0,Y 312.654,Z 611.542,A -85,B 0,C 180,E1 -15464.488,E2 -15464.488} C_VEL
LIN {X 0,Y 312.664,Z 611.541,A -85,B 0,C 180,E1 -15468.329,E2 -15468.329} C_VEL
LIN {X 0,Y 312.865,Z 611.514,A -85,B 0,C 180,E1 -15472.255,E2 -15472.255} C_VEL
LIN {X 0,Y 312.718,Z 611.532,A -85,B 0,C 180,E1 -15474.843,E2 -15474.843} C_VEL
LIN {X 0,Y 312.955,Z 611.503,A -85,B 0,C 180,E1 -15477.426,E2 -15477.426} C_VEL
LIN {X 0,Y 313.113,Z 611.482,A -85,B 0,C 180,E1 -15480.001,E2 -15480.001} C_VEL
LIN {X 0,Y 312.946,Z 611.504,A -85,B 0,C 180,E1 -15482.575,E2 -15482.575} C_VEL
LIN {X 0,Y 312.906,Z 611.505,A -85,B 0,C 180,E1 -15486.449,E2 -15486.449} C_VEL
LIN {X 0,Y 312.781,Z 611.521,A -85,B 0,C 180,E1 -15489.05,E2 -15489.05} C_VEL
LIN {X 0,Y 312.63,Z 611.538,A -85,B 0,C 180,E1 -15492.992,E2 -15492.992} C_VEL
LIN {X 0,Y 312.632,Z 611.535,A -85,B 0,C 180,E1 -15495.651,E2 -15495.651} C_VEL
LIN {X 0,Y 312.625,Z 611.538,A -85,B 0,C 180,E1 -15499.237,E2 -15499.237} C_VEL
LIN {X 0,Y 312.54,Z 611.547,A -85,B 0,C 180,E1 -15502.79,E2 -15502.79} C_VEL
LIN {X 0,Y 312.598,Z 611.538,A -85,B 0,C 180,E1 -15505.937,E2 -15505.937} C_VEL
LIN {X 0,Y 312.542,Z 611.547,A -85,B 0,C 180,E1 -15509.651,E2 -15509.651} C_VEL
LIN {X 0,Y 312.517,Z 611.554,A -85,B 0,C 180,E1 -15513.69,E2 -15513.69} C_VEL
LIN {X 0,Y 312.537,Z 611.55,A -85,B 0,C 180,E1 -15517.384,E2 -15517.384} C_VEL
LIN {X 0,Y 312.498,Z 611.554,A -85,B 0,C 180,E1 -15520.709,E2 -15520.709} C_VEL
LIN {X 0,Y 312.514,Z 611.557,A -85,B 0,C 180,E1 -15524.199,E2 -15524.199} C_VEL
LIN {X 0,Y 312.531,Z 611.554,A -85,B 0,C 180,E1 -15527.91,E2 -15527.91} C_VEL
LIN {X 0,Y 312.543,Z 611.553,A -85,B 0,C 180,E1 -15531.91,E2 -15531.91} C_VEL
LIN {X 0,Y 312.544,Z 611.606,A -85,B 0,C 180,E1 -15533.784,E2 -15533.784} C_VEL
LIN {X 0,Y 314.735,Z 619.99,A -85,B 0,C 180,E1 -15536.834,E2 -15536.834} C_VEL
LIN {X 0,Y 317.218,Z 631.075,A -85,B 0,C 180,E1 -15540.511,E2 -15540.511} C_VEL
LIN {X 0,Y 318.562,Z 638.994,A -85,B 0,C 180,E1 -15542.934,E2 -15542.934} C_VEL
LIN {X 0,Y 318.497,Z 639.564,A -85,B 0,C 180,E1 -15543.086,E2 -15543.086} C_VEL
LIN {X 0,Y 323.007,Z 661.946,A -85,B 0,C 180,E1 -15544.238,E2 -15544.238} C_VEL
LIN {X 0,Y 325.501,Z 679.586,A -85,B 0,C 180,E1 -15544.999,E2 -15544.999} C_VEL
LIN {X 0,Y 326.076,Z 685.413,A -85,B 0,C 180,E1 -15545.219,E2 -15545.219} C_VEL
LIN {X 0,Y 324.015,Z 749.214,A -85,B 0,C 180,E1 -15546.832,E2 -15546.832} C_VEL
LIN {X 0,Y 322.926,Z 763.583,A -85,B 0,C 180,E1 -15547.445,E2 -15547.445} C_VEL
LIN {X 0,Y 321.676,Z 775.59,A -85,B 0,C 180,E1 -15548.198,E2 -15548.198} C_VEL
LIN {X 0,Y 320.056,Z 788.112,A -85,B 0,C 180,E1 -15549.263,E2 -15549.263} C_VEL
LIN {X 0,Y 318.413,Z 799.364,A -85,B 0,C 180,E1 -15550.499,E2 -15550.499} C_VEL
LIN {X 0,Y 316.791,Z 809.575,A -85,B 0,C 180,E1 -15551.906,E2 -15551.906} C_VEL
LIN {X 0,Y 315.231,Z 819.687,A -85,B 0,C 180,E1 -15553.655,E2 -15553.655} C_VEL
LIN {X 0,Y 313.907,Z 827.917,A -85,B 0,C 180,E1 -15555.412,E2 -15555.412} C_VEL
LIN {X 0,Y 312.589,Z 835.244,A -85,B 0,C 180,E1 -15557.338,E2 -15557.338} C_VEL
LIN {X 0,Y 311.868,Z 840.213,A -85,B 0,C 180,E1 -15558.957,E2 -15558.957} C_VEL
LIN {X 0,Y 311.267,Z 845.061,A -85,B 0,C 180,E1 -15560.906,E2 -15560.906} C_VEL
LIN {X 0,Y 310.925,Z 848.785,A -85,B 0,C 180,E1 -15562.859,E2 -15562.859} C_VEL
LIN {X 0,Y 310.77,Z 851.485,A -85,B 0,C 180,E1 -15564.81,E2 -15564.81} C_VEL
LIN {X 0,Y 310.77,Z 852.772,A -85,B 0,C 180,E1 -15566.11,E2 -15566.11} C_VEL
LIN {X 0,Y 310.753,Z 853.603,A -85,B 0,C 180,E1 -15567.408,E2 -15567.408} C_VEL
LIN {X 0,Y 310.784,Z 854.028,A -85,B 0,C 180,E1 -15568.704,E2 -15568.704} C_VEL
LIN {X 0,Y 310.886,Z 854.056,A -85,B 0,C 180,E1 -15570,E2 -15570} C_VEL
LIN {X 0,Y 310.815,Z 853.668,A -85,B 0,C 180,E1 -15571.296,E2 -15571.296} C_VEL
LIN {X 0,Y 310.764,Z 852.821,A -85,B 0,C 180,E1 -15572.592,E2 -15572.592} C_VEL
LIN {X 0,Y 310.793,Z 851.561,A -85,B 0,C 180,E1 -15573.89,E2 -15573.89} C_VEL
LIN {X 0,Y 310.835,Z 848.88,A -85,B 0,C 180,E1 -15575.816,E2 -15575.816} C_VEL
LIN {X 0,Y 311.008,Z 845.053,A -85,B 0,C 180,E1 -15577.792,E2 -15577.792} C_VEL
LIN {X 0,Y 311.388,Z 840.102,A -85,B 0,C 180,E1 -15579.745,E2 -15579.745} C_VEL
LIN {X 0,Y 311.988,Z 833.835,A -85,B 0,C 180,E1 -15581.697,E2 -15581.697} C_VEL
LIN {X 0,Y 313.038,Z 826.022,A -85,B 0,C 180,E1 -15583.635,E2 -15583.635} C_VEL
LIN {X 0,Y 314.014,Z 817.989,A -85,B 0,C 180,E1 -15585.247,E2 -15585.247} C_VEL
LIN {X 0,Y 315.103,Z 808.17,A -85,B 0,C 180,E1 -15586.854,E2 -15586.854} C_VEL
LIN {X 0,Y 316.448,Z 797.3,A -85,B 0,C 180,E1 -15588.282,E2 -15588.282} C_VEL
LIN {X 0,Y 317.68,Z 786.736,A -85,B 0,C 180,E1 -15589.38,E2 -15589.38} C_VEL
LIN {X 0,Y 318.885,Z 774.078,A -85,B 0,C 180,E1 -15590.395,E2 -15590.395} C_VEL
LIN {X 0,Y 319.954,Z 760.812,A -85,B 0,C 180,E1 -15591.165,E2 -15591.165} C_VEL
LIN {X 0,Y 320.609,Z 747.32,A -85,B 0,C 180,E1 -15591.667,E2 -15591.667} C_VEL
LIN {X 0,Y 322.129,Z 682.935,A -85,B 0,C 180,E1 -15593.243,E2 -15593.243} C_VEL
LIN {X 0,Y 316.385,Z 641.894,A -85,B 0,C 180,E1 -15594.718,E2 -15594.718} C_VEL
LIN {X 0,Y 317.239,Z 634.462,A -85,B 0,C 180,E1 -15596.619,E2 -15596.619} C_VEL
LIN {X 0,Y 315.348,Z 624.717,A -85,B 0,C 180,E1 -15599.36,E2 -15599.36} C_VEL
LIN {X 0,Y 312.532,Z 611.555,A -85,B 0,C 180,E1 -15603.264,E2 -15603.264} C_VEL
LIN {X 0,Y 312.54,Z 611.55,A -85,B 0,C 180,E1 -15607.382,E2 -15607.382} C_VEL
LIN {X 0,Y 312.501,Z 611.56,A -85,B 0,C 180,E1 -15610.706,E2 -15610.706} C_VEL
LIN {X 0,Y 312.518,Z 611.556,A -85,B 0,C 180,E1 -15614.196,E2 -15614.196} C_VEL
LIN {X 0,Y 312.527,Z 611.552,A -85,B 0,C 180,E1 -15617.908,E2 -15617.908} C_VEL
LIN {X 0,Y 312.542,Z 611.55,A -85,B 0,C 180,E1 -15621.907,E2 -15621.907} C_VEL
LIN {X 0,Y 312.504,Z 611.555,A -85,B 0,C 180,E1 -15625.789,E2 -15625.789} C_VEL
LIN {X 0,Y 312.525,Z 611.558,A -85,B 0,C 180,E1 -15628.853,E2 -15628.853} C_VEL
LIN {X 0,Y 312.57,Z 611.547,A -85,B 0,C 180,E1 -15631.824,E2 -15631.824} C_VEL
LIN {X 0,Y 312.58,Z 611.548,A -85,B 0,C 180,E1 -15634.71,E2 -15634.71} C_VEL
LIN {X 0,Y 312.531,Z 611.556,A -85,B 0,C 180,E1 -15638.912,E2 -15638.912} C_VEL
LIN {X 0,Y 312.632,Z 611.539,A -85,B 0,C 180,E1 -15641.655,E2 -15641.655} C_VEL
LIN {X 0,Y 312.687,Z 611.534,A -85,B 0,C 180,E1 -15645.685,E2 -15645.685} C_VEL
LIN {X 0,Y 312.694,Z 611.532,A -85,B 0,C 180,E1 -15649.641,E2 -15649.641} C_VEL
LIN {X 0,Y 312.859,Z 611.51,A -85,B 0,C 180,E1 -15652.253,E2 -15652.253} C_VEL
LIN {X 0,Y 312.711,Z 611.53,A -85,B 0,C 180,E1 -15654.842,E2 -15654.842} C_VEL
LIN {X 0,Y 312.985,Z 611.495,A -85,B 0,C 180,E1 -15658.713,E2 -15658.713} C_VEL
LIN {X 0,Y 313.113,Z 611.478,A -85,B 0,C 180,E1 -15659.999,E2 -15659.999} C_VEL
LIN {X 0,Y 312.931,Z 611.5,A -85,B 0,C 180,E1 -15662.574,E2 -15662.574} C_VEL
LIN {X 0,Y 312.886,Z 611.507,A -85,B 0,C 180,E1 -15666.596,E2 -15666.596} C_VEL
LIN {X 0,Y 312.78,Z 611.521,A -85,B 0,C 180,E1 -15669.049,E2 -15669.049} C_VEL
LIN {X 0,Y 312.626,Z 611.538,A -85,B 0,C 180,E1 -15672.991,E2 -15672.991} C_VEL
LIN {X 0,Y 312.63,Z 611.543,A -85,B 0,C 180,E1 -15675.649,E2 -15675.649} C_VEL
LIN {X 0,Y 312.622,Z 611.541,A -85,B 0,C 180,E1 -15679.236,E2 -15679.236} C_VEL
LIN {X 0,Y 312.538,Z 611.549,A -85,B 0,C 180,E1 -15682.789,E2 -15682.789} C_VEL
LIN {X 0,Y 312.595,Z 611.547,A -85,B 0,C 180,E1 -15685.935,E2 -15685.935} C_VEL
LIN {X 0,Y 312.539,Z 611.552,A -85,B 0,C 180,E1 -15689.65,E2 -15689.65} C_VEL
LIN {X 0,Y 312.513,Z 611.556,A -85,B 0,C 180,E1 -15693.689,E2 -15693.689} C_VEL
LIN {X 0,Y 312.545,Z 611.548,A -85,B 0,C 180,E1 -15697.381,E2 -15697.381} C_VEL
LIN {X 0,Y 312.519,Z 611.554,A -85,B 0,C 180,E1 -15700.704,E2 -15700.704} C_VEL
LIN {X 0,Y 312.533,Z 611.557,A -85,B 0,C 180,E1 -15704.194,E2 -15704.194} C_VEL
LIN {X 0,Y 312.527,Z 611.553,A -85,B 0,C 180,E1 -15707.909,E2 -15707.909} C_VEL
LIN {X 0,Y 312.536,Z 611.552,A -85,B 0,C 180,E1 -15711.909,E2 -15711.909} C_VEL
LIN {X 0,Y 312.501,Z 611.556,A -85,B 0,C 180,E1 -15715.79,E2 -15715.79} C_VEL
LIN {X 0,Y 312.515,Z 611.555,A -85,B 0,C 180,E1 -15718.854,E2 -15718.854} C_VEL
LIN {X 0,Y 312.565,Z 611.547,A -85,B 0,C 180,E1 -15721.825,E2 -15721.825} C_VEL
LIN {X 0,Y 312.581,Z 611.55,A -85,B 0,C 180,E1 -15724.711,E2 -15724.711} C_VEL
LIN {X 0,Y 312.583,Z 611.545,A -85,B 0,C 180,E1 -15727.529,E2 -15727.529} C_VEL
LIN {X 0,Y 312.634,Z 611.539,A -85,B 0,C 180,E1 -15731.657,E2 -15731.657} C_VEL
LIN {X 0,Y 312.69,Z 611.531,A -85,B 0,C 180,E1 -15735.686,E2 -15735.686} C_VEL
LIN {X 0,Y 312.698,Z 611.531,A -85,B 0,C 180,E1 -15739.642,E2 -15739.642} C_VEL
LIN {X 0,Y 312.862,Z 611.51,A -85,B 0,C 180,E1 -15742.254,E2 -15742.254} C_VEL
LIN {X 0,Y 312.713,Z 611.533,A -85,B 0,C 180,E1 -15744.842,E2 -15744.842} C_VEL
LIN {X 0,Y 312.988,Z 611.497,A -85,B 0,C 180,E1 -15748.713,E2 -15748.713} C_VEL
LIN {X 0,Y 312.988,Z 611.498,A -85,B 0,C 180,E1 -15751.287,E2 -15751.287} C_VEL
LIN {X 0,Y 312.714,Z 611.534,A -85,B 0,C 180,E1 -15755.158,E2 -15755.158} C_VEL
LIN {X 0,Y 312.85,Z 611.513,A -85,B 0,C 180,E1 -15757.746,E2 -15757.746} C_VEL
LIN {X 0,Y 312.666,Z 611.537,A -85,B 0,C 180,E1 -15761.671,E2 -15761.671} C_VEL
LIN {X 0,Y 312.696,Z 611.533,A -85,B 0,C 180,E1 -15764.887,E2 -15764.887} C_VEL
LIN {X 0,Y 312.643,Z 611.598,A -85,B 0,C 180,E1 -15769.513,E2 -15769.513} C_VEL
LIN {X 0,Y 312.966,Z 613.451,A -85,B 0,C 180,E1 -15770.146,E2 -15770.146} C_VEL
LIN {X 0,Y 322.585,Z 640.289,A -85,B 0,C 180,E1 -15771.528,E2 -15771.528} C_VEL
LIN {X 0,Y 322.939,Z 643.28,A -85,B 0,C 180,E1 -15771.629,E2 -15771.629} C_VEL
LIN {X 0,Y 320.758,Z 720.825,A -85,B 0,C 180,E1 -15773.527,E2 -15773.527} C_VEL
LIN {X 0,Y 320.119,Z 734.67,A -85,B 0,C 180,E1 -15774.135,E2 -15774.135} C_VEL
LIN {X 0,Y 319.232,Z 747.465,A -85,B 0,C 180,E1 -15774.963,E2 -15774.963} C_VEL
LIN {X 0,Y 318.241,Z 758.919,A -85,B 0,C 180,E1 -15775.96,E2 -15775.96} C_VEL
LIN {X 0,Y 317.029,Z 770.418,A -85,B 0,C 180,E1 -15777.235,E2 -15777.235} C_VEL
LIN {X 0,Y 315.889,Z 780.107,A -85,B 0,C 180,E1 -15778.576,E2 -15778.576} C_VEL
LIN {X 0,Y 314.755,Z 789.664,A -85,B 0,C 180,E1 -15780.219,E2 -15780.219} C_VEL
LIN {X 0,Y 313.606,Z 798.395,A -85,B 0,C 180,E1 -15782.073,E2 -15782.073} C_VEL
LIN {X 0,Y 312.776,Z 804.844,A -85,B 0,C 180,E1 -15783.761,E2 -15783.761} C_VEL
LIN {X 0,Y 311.997,Z 811.27,A -85,B 0,C 180,E1 -15785.849,E2 -15785.849} C_VEL
LIN {X 0,Y 311.443,Z 815.987,A -85,B 0,C 180,E1 -15787.834,E2 -15787.834} C_VEL
LIN {X 0,Y 311.038,Z 819.53,A -85,B 0,C 180,E1 -15789.805,E2 -15789.805} C_VEL
LIN {X 0,Y 310.759,Z 821.988,A -85,B 0,C 180,E1 -15791.729,E2 -15791.729} C_VEL
LIN {X 0,Y 310.619,Z 823.48,A -85,B 0,C 180,E1 -15793.613,E2 -15793.613} C_VEL
LIN {X 0,Y 310.57,Z 824.096,A -85,B 0,C 180,E1 -15795.453,E2 -15795.453} C_VEL
LIN {X 0,Y 310.682,Z 823.918,A -85,B 0,C 180,E1 -15797.264,E2 -15797.264} C_VEL
LIN {X 0,Y 310.936,Z 822.989,A -85,B 0,C 180,E1 -15799.045,E2 -15799.045} C_VEL
LIN {X 0,Y 311.298,Z 821.309,A -85,B 0,C 180,E1 -15800.793,E2 -15800.793} C_VEL
LIN {X 0,Y 311.726,Z 818.896,A -85,B 0,C 180,E1 -15802.503,E2 -15802.503} C_VEL
LIN {X 0,Y 312.294,Z 815.757,A -85,B 0,C 180,E1 -15804.19,E2 -15804.19} C_VEL
LIN {X 0,Y 313.156,Z 811.065,A -85,B 0,C 180,E1 -15806.135,E2 -15806.135} C_VEL
LIN {X 0,Y 314.318,Z 804.759,A -85,B 0,C 180,E1 -15808.173,E2 -15808.173} C_VEL
LIN {X 0,Y 314.477,Z 803.853,A -85,B 0,C 180,E1 -15808.428,E2 -15808.428} C_VEL
LIN {X 0,Y 314.446,Z 800.652,A -85,B 0,C 180,E1 -15809.335,E2 -15809.335} C_VEL
LIN {X 0,Y 312.796,Z 795.238,A -85,B 0,C 180,E1 -15810.825,E2 -15810.825} C_VEL
LIN {X 0,Y 311.202,Z 789.236,A -85,B 0,C 180,E1 -15812.243,E2 -15812.243} C_VEL
LIN {X 0,Y 311.241,Z 785.116,A -85,B 0,C 180,E1 -15813.022,E2 -15813.022} C_VEL
LIN {X 0,Y 312.949,Z 774.76,A -85,B 0,C 180,E1 -15814.604,E2 -15814.604} C_VEL
LIN {X 0,Y 314.311,Z 765.405,A -85,B 0,C 180,E1 -15815.76,E2 -15815.76} C_VEL
LIN {X 0,Y 315.806,Z 753.777,A -85,B 0,C 180,E1 -15816.907,E2 -15816.907} C_VEL
LIN {X 0,Y 317.091,Z 740.791,A -85,B 0,C 180,E1 -15817.866,E2 -15817.866} C_VEL
LIN {X 0,Y 317.942,Z 727.919,A -85,B 0,C 180,E1 -15818.553,E2 -15818.553} C_VEL
LIN {X 0,Y 318.611,Z 713.88,A -85,B 0,C 180,E1 -15819.004,E2 -15819.004} C_VEL
LIN {X 0,Y 320.993,Z 647.341,A -85,B 0,C 180,E1 -15820.704,E2 -15820.704} C_VEL
LIN {X 0,Y 314.461,Z 632.239,A -85,B 0,C 180,E1 -15821.894,E2 -15821.894} C_VEL
LIN {X 0,Y 308.41,Z 620.202,A -85,B 0,C 180,E1 -15823.018,E2 -15823.018} C_VEL
LIN {X 0,Y 306.611,Z 616.651,A -85,B 0,C 180,E1 -15823.395,E2 -15823.395} C_VEL
LIN {X 0,Y 305.637,Z 612.415,A -85,B 0,C 180,E1 -15825.26,E2 -15825.26} C_VEL
LIN {X 0,Y 305.633,Z 612.416,A -85,B 0,C 180,E1 -15829.4,E2 -15829.4} C_VEL
LIN {X 0,Y 305.806,Z 612.394,A -85,B 0,C 180,E1 -15832.075,E2 -15832.075} C_VEL
LIN {X 0,Y 305.689,Z 612.407,A -85,B 0,C 180,E1 -15834.724,E2 -15834.724} C_VEL
LIN {X 0,Y 305.955,Z 612.372,A -85,B 0,C 180,E1 -15838.684,E2 -15838.684} C_VEL
LIN {X 0,Y 305.954,Z 612.371,A -85,B 0,C 180,E1 -15841.317,E2 -15841.317} C_VEL
LIN {X 0,Y 305.687,Z 612.409,A -85,B 0,C 180,E1 -15845.277,E2 -15845.277} C_VEL
LIN {X 0,Y 305.807,Z 612.392,A -85,B 0,C 180,E1 -15847.926,E2 -15847.926} C_VEL
LIN {X 0,Y 305.6,Z 612.416,A -85,B 0,C 180,E1 -15851.946,E2 -15851.946} C_VEL
LIN {X 0,Y 305.632,Z 612.412,A -85,B 0,C 180,E1 -15855.036,E2 -15855.036} C_VEL
LIN {X 0,Y 305.571,Z 612.417,A -85,B 0,C 180,E1 -15859.446,E2 -15859.446} C_VEL
LIN {X 0,Y 305.485,Z 612.427,A -85,B 0,C 180,E1 -15863.042,E2 -15863.042} C_VEL
LIN {X 0,Y 305.543,Z 612.418,A -85,B 0,C 180,E1 -15866.228,E2 -15866.228} C_VEL
